KUKA KRL program: Robotarmmovement.src

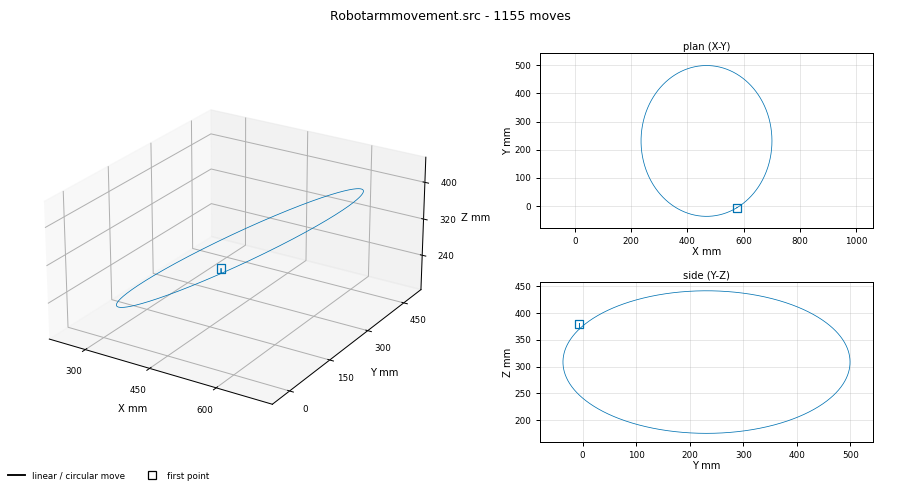
[picture p0: tool path of Robotarmmovement.src, 1155 of 1157 moves have a stored position in this frame; points joined in program order, loops and branches not executed]
&ACCESS RVP
&PARAM EDITMASK = *
&PARAM TEMPLATE = C:\KRC\Roboter\Template\vorgabe
DEF Robotarmmovement( )


;FOLD INI
;FOLD BASISTECH INI
GLOBAL INTERRUPT DECL 3 WHEN $STOPMESS==TRUE DO IR_STOPM ( )
INTERRUPT ON 3
BAS (#INITMOV,0 )
;ENDFOLD (BASISTECH INI)
;ENDFOLD (INI)

;FOLD STARTPOSITION - BASE IS 0, TOOL IS 6, SPEED IS 15%, POSITION IS A1 5,A2 -90,A3 100,A4 5,A5 -10,A6 -5,E1 0,E2 0,E3 0,E4 0
$BWDSTART = FALSE
PDAT_ACT = {VEL 15,ACC 100,APO_DIST 50}
FDAT_ACT = {TOOL_NO 6,BASE_NO 0,IPO_FRAME #BASE}
BAS (#PTP_PARAMS,15)
PTP  {A1 5,A2 -90,A3 100,A4 5,A5 -10,A6 -5,E1 0,E2 0,E3 0,E4 0}
;ENDFOLD

;FOLD LIN SPEED IS 0.25 m/sec, INTERPOLATION SETTINGS IN FOLD
$VEL.CP=0.25
$ADVANCE=3
;ENDFOLD

;FOLD COMMANDS IN FOLD. SELECT EDIT/FOLDS/OPEN ALL FOLDS TO DISPLAY
PTP {X 576.159, Y -6.053, Z 380.301, A 0, B 90, C -61.802, E1 0, E2 0, E3 0, E4 0, S 'B 110'} C_PTP
LIN {X 576.159, Y -6.053, Z 380.301, A 0, B 90, C -61.802, E1 0, E2 0, E3 0, E4 0}
LIN {X 576.159, Y -6.053, Z 370.301, A 0, B 90, C -61.802, E1 0, E2 0, E3 0, E4 0} C_DIS
LIN {X 577.282, Y -5.37, Z 370.943, A 0, B 90, C -61.726, E1 0, E2 0, E3 0, E4 0} C_DIS
LIN {X 578.402, Y -4.68, Z 371.584, A 0, B 90, C -61.652, E1 0, E2 0, E3 0, E4 0} C_DIS
LIN {X 579.519, Y -3.984, Z 372.223, A 0, B 90, C -61.578, E1 0, E2 0, E3 0, E4 0} C_DIS
LIN {X 580.632, Y -3.28, Z 372.86, A 0, B 90, C -61.506, E1 0, E2 0, E3 0, E4 0} C_DIS
LIN {X 581.742, Y -2.569, Z 373.495, A 0, B 90, C -61.434, E1 0, E2 0, E3 0, E4 0} C_DIS
LIN {X 582.848, Y -1.851, Z 374.128, A 0, B 90, C -61.364, E1 0, E2 0, E3 0, E4 0} C_DIS
LIN {X 583.952, Y -1.126, Z 374.759, A 0, B 90, C -61.294, E1 0, E2 0, E3 0, E4 0} C_DIS
LIN {X 585.051, Y -0.395, Z 375.389, A 0, B 90, C -61.226, E1 0, E2 0, E3 0, E4 0} C_DIS
LIN {X 586.148, Y 0.344, Z 376.016, A 0, B 90, C -61.159, E1 0, E2 0, E3 0, E4 0} C_DIS
LIN {X 587.24, Y 1.089, Z 376.641, A 0, B 90, C -61.093, E1 0, E2 0, E3 0, E4 0} C_DIS
LIN {X 588.329, Y 1.842, Z 377.264, A 0, B 90, C -61.027, E1 0, E2 0, E3 0, E4 0} C_DIS
LIN {X 589.415, Y 2.601, Z 377.885, A 0, B 90, C -60.963, E1 0, E2 0, E3 0, E4 0} C_DIS
LIN {X 590.497, Y 3.367, Z 378.504, A 0, B 90, C -60.9, E1 0, E2 0, E3 0, E4 0} C_DIS
LIN {X 591.575, Y 4.14, Z 379.121, A 0, B 90, C -60.838, E1 0, E2 0, E3 0, E4 0} C_DIS
LIN {X 592.65, Y 4.919, Z 379.736, A 0, B 90, C -60.776, E1 0, E2 0, E3 0, E4 0} C_DIS
LIN {X 593.721, Y 5.705, Z 380.349, A 0, B 90, C -60.716, E1 0, E2 0, E3 0, E4 0} C_DIS
LIN {X 594.788, Y 6.498, Z 380.96, A 0, B 90, C -60.657, E1 0, E2 0, E3 0, E4 0} C_DIS
LIN {X 595.851, Y 7.298, Z 381.568, A 0, B 90, C -60.598, E1 0, E2 0, E3 0, E4 0} C_DIS
LIN {X 596.911, Y 8.105, Z 382.174, A 0, B 90, C -60.541, E1 0, E2 0, E3 0, E4 0} C_DIS
LIN {X 597.967, Y 8.918, Z 382.778, A 0, B 90, C -60.485, E1 0, E2 0, E3 0, E4 0} C_DIS
LIN {X 599.019, Y 9.737, Z 383.38, A 0, B 90, C -60.43, E1 0, E2 0, E3 0, E4 0} C_DIS
LIN {X 600.067, Y 10.564, Z 383.98, A 0, B 90, C -60.375, E1 0, E2 0, E3 0, E4 0} C_DIS
LIN {X 601.111, Y 11.396, Z 384.577, A 0, B 90, C -60.322, E1 0, E2 0, E3 0, E4 0} C_DIS
LIN {X 602.151, Y 12.236, Z 385.172, A 0, B 90, C -60.269, E1 0, E2 0, E3 0, E4 0} C_DIS
LIN {X 603.187, Y 13.082, Z 385.765, A 0, B 90, C -60.218, E1 0, E2 0, E3 0, E4 0} C_DIS
LIN {X 604.219, Y 13.934, Z 386.356, A 0, B 90, C -60.167, E1 0, E2 0, E3 0, E4 0} C_DIS
LIN {X 605.247, Y 14.793, Z 386.944, A 0, B 90, C -60.118, E1 0, E2 0, E3 0, E4 0} C_DIS
LIN {X 606.271, Y 15.658, Z 387.53, A 0, B 90, C -60.069, E1 0, E2 0, E3 0, E4 0} C_DIS
LIN {X 607.291, Y 16.53, Z 388.113, A 0, B 90, C -60.022, E1 0, E2 0, E3 0, E4 0} C_DIS
LIN {X 608.307, Y 17.408, Z 388.695, A 0, B 90, C -59.975, E1 0, E2 0, E3 0, E4 0} C_DIS
LIN {X 609.318, Y 18.293, Z 389.273, A 0, B 90, C -59.929, E1 0, E2 0, E3 0, E4 0} C_DIS
LIN {X 610.325, Y 19.184, Z 389.85, A 0, B 90, C -59.884, E1 0, E2 0, E3 0, E4 0} C_DIS
LIN {X 611.328, Y 20.081, Z 390.424, A 0, B 90, C -59.84, E1 0, E2 0, E3 0, E4 0} C_DIS
LIN {X 612.327, Y 20.985, Z 390.995, A 0, B 90, C -59.798, E1 0, E2 0, E3 0, E4 0} C_DIS
LIN {X 613.322, Y 21.895, Z 391.564, A 0, B 90, C -59.755, E1 0, E2 0, E3 0, E4 0} C_DIS
LIN {X 614.312, Y 22.811, Z 392.131, A 0, B 90, C -59.714, E1 0, E2 0, E3 0, E4 0} C_DIS
LIN {X 615.298, Y 23.733, Z 392.695, A 0, B 90, C -59.674, E1 0, E2 0, E3 0, E4 0} C_DIS
LIN {X 616.279, Y 24.661, Z 393.256, A 0, B 90, C -59.635, E1 0, E2 0, E3 0, E4 0} C_DIS
LIN {X 617.256, Y 25.596, Z 393.815, A 0, B 90, C -59.596, E1 0, E2 0, E3 0, E4 0} C_DIS
LIN {X 618.229, Y 26.537, Z 394.372, A 0, B 90, C -59.559, E1 0, E2 0, E3 0, E4 0} C_DIS
LIN {X 619.197, Y 27.483, Z 394.926, A 0, B 90, C -59.522, E1 0, E2 0, E3 0, E4 0} C_DIS
LIN {X 620.161, Y 28.436, Z 395.477, A 0, B 90, C -59.486, E1 0, E2 0, E3 0, E4 0} C_DIS
LIN {X 621.12, Y 29.395, Z 396.026, A 0, B 90, C -59.452, E1 0, E2 0, E3 0, E4 0} C_DIS
LIN {X 622.074, Y 30.36, Z 396.572, A 0, B 90, C -59.418, E1 0, E2 0, E3 0, E4 0} C_DIS
LIN {X 623.024, Y 31.331, Z 397.116, A 0, B 90, C -59.385, E1 0, E2 0, E3 0, E4 0} C_DIS
LIN {X 623.97, Y 32.308, Z 397.657, A 0, B 90, C -59.352, E1 0, E2 0, E3 0, E4 0} C_DIS
LIN {X 624.91, Y 33.291, Z 398.195, A 0, B 90, C -59.321, E1 0, E2 0, E3 0, E4 0} C_DIS
LIN {X 625.846, Y 34.28, Z 398.73, A 0, B 90, C -59.29, E1 0, E2 0, E3 0, E4 0} C_DIS
LIN {X 626.778, Y 35.274, Z 399.263, A 0, B 90, C -59.261, E1 0, E2 0, E3 0, E4 0} C_DIS
LIN {X 627.704, Y 36.275, Z 399.793, A 0, B 90, C -59.232, E1 0, E2 0, E3 0, E4 0} C_DIS
LIN {X 628.626, Y 37.281, Z 400.321, A 0, B 90, C -59.204, E1 0, E2 0, E3 0, E4 0} C_DIS
LIN {X 629.543, Y 38.293, Z 400.846, A 0, B 90, C -59.177, E1 0, E2 0, E3 0, E4 0} C_DIS
LIN {X 630.455, Y 39.311, Z 401.368, A 0, B 90, C -59.151, E1 0, E2 0, E3 0, E4 0} C_DIS
LIN {X 631.363, Y 40.335, Z 401.887, A 0, B 90, C -59.125, E1 0, E2 0, E3 0, E4 0} C_DIS
LIN {X 632.265, Y 41.364, Z 402.403, A 0, B 90, C -59.101, E1 0, E2 0, E3 0, E4 0} C_DIS
LIN {X 633.163, Y 42.399, Z 402.917, A 0, B 90, C -59.077, E1 0, E2 0, E3 0, E4 0} C_DIS
LIN {X 634.056, Y 43.439, Z 403.428, A 0, B 90, C -59.054, E1 0, E2 0, E3 0, E4 0} C_DIS
LIN {X 634.943, Y 44.485, Z 403.936, A 0, B 90, C -59.032, E1 0, E2 0, E3 0, E4 0} C_DIS
LIN {X 635.826, Y 45.537, Z 404.441, A 0, B 90, C -59.01, E1 0, E2 0, E3 0, E4 0} C_DIS
LIN {X 636.704, Y 46.594, Z 404.943, A 0, B 90, C -58.99, E1 0, E2 0, E3 0, E4 0} C_DIS
LIN {X 637.577, Y 47.657, Z 405.442, A 0, B 90, C -58.97, E1 0, E2 0, E3 0, E4 0} C_DIS
LIN {X 638.445, Y 48.725, Z 405.939, A 0, B 90, C -58.951, E1 0, E2 0, E3 0, E4 0} C_DIS
LIN {X 639.307, Y 49.799, Z 406.432, A 0, B 90, C -58.933, E1 0, E2 0, E3 0, E4 0} C_DIS
LIN {X 640.165, Y 50.878, Z 406.923, A 0, B 90, C -58.916, E1 0, E2 0, E3 0, E4 0} C_DIS
LIN {X 641.017, Y 51.962, Z 407.411, A 0, B 90, C -58.899, E1 0, E2 0, E3 0, E4 0} C_DIS
LIN {X 641.865, Y 53.052, Z 407.896, A 0, B 90, C -58.883, E1 0, E2 0, E3 0, E4 0} C_DIS
LIN {X 642.707, Y 54.147, Z 408.378, A 0, B 90, C -58.868, E1 0, E2 0, E3 0, E4 0} C_DIS
LIN {X 643.544, Y 55.248, Z 408.856, A 0, B 90, C -58.854, E1 0, E2 0, E3 0, E4 0} C_DIS
LIN {X 644.375, Y 56.353, Z 409.332, A 0, B 90, C -58.84, E1 0, E2 0, E3 0, E4 0} C_DIS
LIN {X 645.202, Y 57.464, Z 409.805, A 0, B 90, C -58.828, E1 0, E2 0, E3 0, E4 0} C_DIS
LIN {X 646.023, Y 58.58, Z 410.275, A 0, B 90, C -58.816, E1 0, E2 0, E3 0, E4 0} C_DIS
LIN {X 646.839, Y 59.701, Z 410.742, A 0, B 90, C -58.804, E1 0, E2 0, E3 0, E4 0} C_DIS
LIN {X 647.65, Y 60.828, Z 411.206, A 0, B 90, C -58.794, E1 0, E2 0, E3 0, E4 0} C_DIS
LIN {X 648.455, Y 61.959, Z 411.666, A 0, B 90, C -58.784, E1 0, E2 0, E3 0, E4 0} C_DIS
LIN {X 649.255, Y 63.095, Z 412.124, A 0, B 90, C -58.775, E1 0, E2 0, E3 0, E4 0} C_DIS
LIN {X 650.049, Y 64.237, Z 412.579, A 0, B 90, C -58.767, E1 0, E2 0, E3 0, E4 0} C_DIS
LIN {X 650.838, Y 65.383, Z 413.03, A 0, B 90, C -58.759, E1 0, E2 0, E3 0, E4 0} C_DIS
LIN {X 651.622, Y 66.535, Z 413.478, A 0, B 90, C -58.752, E1 0, E2 0, E3 0, E4 0} C_DIS
LIN {X 652.4, Y 67.691, Z 413.924, A 0, B 90, C -58.746, E1 0, E2 0, E3 0, E4 0} C_DIS
LIN {X 653.172, Y 68.852, Z 414.366, A 0, B 90, C -58.74, E1 0, E2 0, E3 0, E4 0} C_DIS
LIN {X 653.94, Y 70.018, Z 414.805, A 0, B 90, C -58.736, E1 0, E2 0, E3 0, E4 0} C_DIS
LIN {X 654.701, Y 71.189, Z 415.24, A 0, B 90, C -58.732, E1 0, E2 0, E3 0, E4 0} C_DIS
LIN {X 655.457, Y 72.364, Z 415.673, A 0, B 90, C -58.728, E1 0, E2 0, E3 0, E4 0} C_DIS
LIN {X 656.208, Y 73.545, Z 416.102, A 0, B 90, C -58.726, E1 0, E2 0, E3 0, E4 0} C_DIS
LIN {X 656.952, Y 74.73, Z 416.529, A 0, B 90, C -58.724, E1 0, E2 0, E3 0, E4 0} C_DIS
LIN {X 657.692, Y 75.919, Z 416.951, A 0, B 90, C -58.722, E1 0, E2 0, E3 0, E4 0} C_DIS
LIN {X 658.425, Y 77.114, Z 417.371, A 0, B 90, C -58.722, E1 0, E2 0, E3 0, E4 0} C_DIS
LIN {X 659.153, Y 78.313, Z 417.788, A 0, B 90, C -58.722, E1 0, E2 0, E3 0, E4 0} C_DIS
LIN {X 659.875, Y 79.516, Z 418.201, A 0, B 90, C -58.722, E1 0, E2 0, E3 0, E4 0} C_DIS
LIN {X 660.592, Y 80.724, Z 418.611, A 0, B 90, C -58.724, E1 0, E2 0, E3 0, E4 0} C_DIS
LIN {X 661.302, Y 81.936, Z 419.017, A 0, B 90, C -58.726, E1 0, E2 0, E3 0, E4 0} C_DIS
LIN {X 662.007, Y 83.153, Z 419.421, A 0, B 90, C -58.728, E1 0, E2 0, E3 0, E4 0} C_DIS
LIN {X 662.707, Y 84.375, Z 419.821, A 0, B 90, C -58.732, E1 0, E2 0, E3 0, E4 0} C_DIS
LIN {X 663.4, Y 85.6, Z 420.218, A 0, B 90, C -58.736, E1 0, E2 0, E3 0, E4 0} C_DIS
LIN {X 664.088, Y 86.83, Z 420.611, A 0, B 90, C -58.74, E1 0, E2 0, E3 0, E4 0} C_DIS
LIN {X 664.769, Y 88.065, Z 421.001, A 0, B 90, C -58.746, E1 0, E2 0, E3 0, E4 0} C_DIS
LIN {X 665.445, Y 89.303, Z 421.388, A 0, B 90, C -58.751, E1 0, E2 0, E3 0, E4 0} C_DIS
LIN {X 666.115, Y 90.546, Z 421.771, A 0, B 90, C -58.758, E1 0, E2 0, E3 0, E4 0} C_DIS
LIN {X 666.779, Y 91.793, Z 422.151, A 0, B 90, C -58.765, E1 0, E2 0, E3 0, E4 0} C_DIS
LIN {X 667.438, Y 93.045, Z 422.528, A 0, B 90, C -58.773, E1 0, E2 0, E3 0, E4 0} C_DIS
LIN {X 668.09, Y 94.3, Z 422.901, A 0, B 90, C -58.781, E1 0, E2 0, E3 0, E4 0} C_DIS
LIN {X 668.736, Y 95.559, Z 423.271, A 0, B 90, C -58.79, E1 0, E2 0, E3 0, E4 0} C_DIS
LIN {X 669.376, Y 96.823, Z 423.637, A 0, B 90, C -58.8, E1 0, E2 0, E3 0, E4 0} C_DIS
LIN {X 670.011, Y 98.09, Z 424, A 0, B 90, C -58.81, E1 0, E2 0, E3 0, E4 0} C_DIS
LIN {X 670.639, Y 99.362, Z 424.36, A 0, B 90, C -58.821, E1 0, E2 0, E3 0, E4 0} C_DIS
LIN {X 671.261, Y 100.637, Z 424.716, A 0, B 90, C -58.832, E1 0, E2 0, E3 0, E4 0} C_DIS
LIN {X 671.878, Y 101.916, Z 425.068, A 0, B 90, C -58.844, E1 0, E2 0, E3 0, E4 0} C_DIS
LIN {X 672.488, Y 103.199, Z 425.418, A 0, B 90, C -58.856, E1 0, E2 0, E3 0, E4 0} C_DIS
LIN {X 673.092, Y 104.486, Z 425.763, A 0, B 90, C -58.87, E1 0, E2 0, E3 0, E4 0} C_DIS
LIN {X 673.69, Y 105.777, Z 426.105, A 0, B 90, C -58.883, E1 0, E2 0, E3 0, E4 0} C_DIS
LIN {X 674.282, Y 107.072, Z 426.444, A 0, B 90, C -58.898, E1 0, E2 0, E3 0, E4 0} C_DIS
LIN {X 674.867, Y 108.37, Z 426.779, A 0, B 90, C -58.912, E1 0, E2 0, E3 0, E4 0} C_DIS
LIN {X 675.447, Y 109.672, Z 427.111, A 0, B 90, C -58.928, E1 0, E2 0, E3 0, E4 0} C_DIS
LIN {X 676.02, Y 110.977, Z 427.439, A 0, B 90, C -58.944, E1 0, E2 0, E3 0, E4 0} C_DIS
LIN {X 676.588, Y 112.286, Z 427.763, A 0, B 90, C -58.96, E1 0, E2 0, E3 0, E4 0} C_DIS
LIN {X 677.148, Y 113.599, Z 428.084, A 0, B 90, C -58.977, E1 0, E2 0, E3 0, E4 0} C_DIS
LIN {X 677.703, Y 114.915, Z 428.402, A 0, B 90, C -58.995, E1 0, E2 0, E3 0, E4 0} C_DIS
LIN {X 678.252, Y 116.234, Z 428.715, A 0, B 90, C -59.013, E1 0, E2 0, E3 0, E4 0} C_DIS
LIN {X 678.794, Y 117.557, Z 429.026, A 0, B 90, C -59.032, E1 0, E2 0, E3 0, E4 0} C_DIS
LIN {X 679.33, Y 118.884, Z 429.332, A 0, B 90, C -59.051, E1 0, E2 0, E3 0, E4 0} C_DIS
LIN {X 679.859, Y 120.214, Z 429.635, A 0, B 90, C -59.071, E1 0, E2 0, E3 0, E4 0} C_DIS
LIN {X 680.383, Y 121.547, Z 429.935, A 0, B 90, C -59.091, E1 0, E2 0, E3 0, E4 0} C_DIS
LIN {X 680.9, Y 122.883, Z 430.231, A 0, B 90, C -59.112, E1 0, E2 0, E3 0, E4 0} C_DIS
LIN {X 681.411, Y 124.222, Z 430.523, A 0, B 90, C -59.133, E1 0, E2 0, E3 0, E4 0} C_DIS
LIN {X 681.915, Y 125.565, Z 430.811, A 0, B 90, C -59.155, E1 0, E2 0, E3 0, E4 0} C_DIS
LIN {X 682.413, Y 126.911, Z 431.096, A 0, B 90, C -59.177, E1 0, E2 0, E3 0, E4 0} C_DIS
LIN {X 682.904, Y 128.26, Z 431.378, A 0, B 90, C -59.2, E1 0, E2 0, E3 0, E4 0} C_DIS
LIN {X 683.39, Y 129.612, Z 431.655, A 0, B 90, C -59.224, E1 0, E2 0, E3 0, E4 0} C_DIS
LIN {X 683.868, Y 130.967, Z 431.929, A 0, B 90, C -59.247, E1 0, E2 0, E3 0, E4 0} C_DIS
LIN {X 684.341, Y 132.325, Z 432.199, A 0, B 90, C -59.272, E1 0, E2 0, E3 0, E4 0} C_DIS
LIN {X 684.807, Y 133.687, Z 432.466, A 0, B 90, C -59.297, E1 0, E2 0, E3 0, E4 0} C_DIS
LIN {X 685.266, Y 135.051, Z 432.729, A 0, B 90, C -59.322, E1 0, E2 0, E3 0, E4 0} C_DIS
LIN {X 685.719, Y 136.417, Z 432.988, A 0, B 90, C -59.348, E1 0, E2 0, E3 0, E4 0} C_DIS
LIN {X 686.166, Y 137.787, Z 433.244, A 0, B 90, C -59.374, E1 0, E2 0, E3 0, E4 0} C_DIS
LIN {X 686.606, Y 139.159, Z 433.495, A 0, B 90, C -59.401, E1 0, E2 0, E3 0, E4 0} C_DIS
LIN {X 687.039, Y 140.535, Z 433.743, A 0, B 90, C -59.428, E1 0, E2 0, E3 0, E4 0} C_DIS
LIN {X 687.466, Y 141.913, Z 433.988, A 0, B 90, C -59.456, E1 0, E2 0, E3 0, E4 0} C_DIS
LIN {X 687.886, Y 143.293, Z 434.228, A 0, B 90, C -59.484, E1 0, E2 0, E3 0, E4 0} C_DIS
LIN {X 688.3, Y 144.676, Z 434.465, A 0, B 90, C -59.513, E1 0, E2 0, E3 0, E4 0} C_DIS
LIN {X 688.708, Y 146.062, Z 434.698, A 0, B 90, C -59.542, E1 0, E2 0, E3 0, E4 0} C_DIS
LIN {X 689.108, Y 147.45, Z 434.927, A 0, B 90, C -59.571, E1 0, E2 0, E3 0, E4 0} C_DIS
LIN {X 689.503, Y 148.841, Z 435.153, A 0, B 90, C -59.601, E1 0, E2 0, E3 0, E4 0} C_DIS
LIN {X 689.89, Y 150.235, Z 435.375, A 0, B 90, C -59.632, E1 0, E2 0, E3 0, E4 0} C_DIS
LIN {X 690.271, Y 151.63, Z 435.593, A 0, B 90, C -59.663, E1 0, E2 0, E3 0, E4 0} C_DIS
LIN {X 690.645, Y 153.028, Z 435.807, A 0, B 90, C -59.694, E1 0, E2 0, E3 0, E4 0} C_DIS
LIN {X 691.013, Y 154.429, Z 436.017, A 0, B 90, C -59.726, E1 0, E2 0, E3 0, E4 0} C_DIS
LIN {X 691.374, Y 155.831, Z 436.224, A 0, B 90, C -59.758, E1 0, E2 0, E3 0, E4 0} C_DIS
LIN {X 691.729, Y 157.236, Z 436.427, A 0, B 90, C -59.791, E1 0, E2 0, E3 0, E4 0} C_DIS
LIN {X 692.076, Y 158.643, Z 436.626, A 0, B 90, C -59.824, E1 0, E2 0, E3 0, E4 0} C_DIS
LIN {X 692.417, Y 160.053, Z 436.821, A 0, B 90, C -59.858, E1 0, E2 0, E3 0, E4 0} C_DIS
LIN {X 692.752, Y 161.464, Z 437.012, A 0, B 90, C -59.892, E1 0, E2 0, E3 0, E4 0} C_DIS
LIN {X 693.08, Y 162.878, Z 437.2, A 0, B 90, C -59.926, E1 0, E2 0, E3 0, E4 0} C_DIS
LIN {X 693.401, Y 164.293, Z 437.383, A 0, B 90, C -59.961, E1 0, E2 0, E3 0, E4 0} C_DIS
LIN {X 693.715, Y 165.711, Z 437.563, A 0, B 90, C -59.996, E1 0, E2 0, E3 0, E4 0} C_DIS
LIN {X 694.022, Y 167.13, Z 437.739, A 0, B 90, C -60.032, E1 0, E2 0, E3 0, E4 0} C_DIS
LIN {X 694.323, Y 168.552, Z 437.911, A 0, B 90, C -60.068, E1 0, E2 0, E3 0, E4 0} C_DIS
LIN {X 694.617, Y 169.975, Z 438.079, A 0, B 90, C -60.104, E1 0, E2 0, E3 0, E4 0} C_DIS
LIN {X 694.905, Y 171.4, Z 438.244, A 0, B 90, C -60.141, E1 0, E2 0, E3 0, E4 0} C_DIS
LIN {X 695.185, Y 172.827, Z 438.404, A 0, B 90, C -60.178, E1 0, E2 0, E3 0, E4 0} C_DIS
LIN {X 695.459, Y 174.256, Z 438.561, A 0, B 90, C -60.216, E1 0, E2 0, E3 0, E4 0} C_DIS
LIN {X 695.726, Y 175.686, Z 438.714, A 0, B 90, C -60.254, E1 0, E2 0, E3 0, E4 0} C_DIS
LIN {X 695.987, Y 177.118, Z 438.863, A 0, B 90, C -60.292, E1 0, E2 0, E3 0, E4 0} C_DIS
LIN {X 696.24, Y 178.552, Z 439.008, A 0, B 90, C -60.331, E1 0, E2 0, E3 0, E4 0} C_DIS
LIN {X 696.487, Y 179.987, Z 439.149, A 0, B 90, C -60.37, E1 0, E2 0, E3 0, E4 0} C_DIS
LIN {X 696.727, Y 181.424, Z 439.286, A 0, B 90, C -60.409, E1 0, E2 0, E3 0, E4 0} C_DIS
LIN {X 696.96, Y 182.862, Z 439.42, A 0, B 90, C -60.449, E1 0, E2 0, E3 0, E4 0} C_DIS
LIN {X 697.186, Y 184.302, Z 439.549, A 0, B 90, C -60.49, E1 0, E2 0, E3 0, E4 0} C_DIS
LIN {X 697.405, Y 185.743, Z 439.675, A 0, B 90, C -60.53, E1 0, E2 0, E3 0, E4 0} C_DIS
LIN {X 697.618, Y 187.185, Z 439.796, A 0, B 90, C -60.571, E1 0, E2 0, E3 0, E4 0} C_DIS
LIN {X 697.824, Y 188.629, Z 439.914, A 0, B 90, C -60.613, E1 0, E2 0, E3 0, E4 0} C_DIS
LIN {X 698.023, Y 190.074, Z 440.028, A 0, B 90, C -60.654, E1 0, E2 0, E3 0, E4 0} C_DIS
LIN {X 698.215, Y 191.52, Z 440.138, A 0, B 90, C -60.696, E1 0, E2 0, E3 0, E4 0} C_DIS
LIN {X 698.4, Y 192.968, Z 440.244, A 0, B 90, C -60.739, E1 0, E2 0, E3 0, E4 0} C_DIS
LIN {X 698.578, Y 194.416, Z 440.346, A 0, B 90, C -60.782, E1 0, E2 0, E3 0, E4 0} C_DIS
LIN {X 698.75, Y 195.866, Z 440.444, A 0, B 90, C -60.825, E1 0, E2 0, E3 0, E4 0} C_DIS
LIN {X 698.914, Y 197.317, Z 440.538, A 0, B 90, C -60.868, E1 0, E2 0, E3 0, E4 0} C_DIS
LIN {X 699.072, Y 198.768, Z 440.628, A 0, B 90, C -60.912, E1 0, E2 0, E3 0, E4 0} C_DIS
LIN {X 699.223, Y 200.221, Z 440.715, A 0, B 90, C -60.956, E1 0, E2 0, E3 0, E4 0} C_DIS
LIN {X 699.367, Y 201.675, Z 440.797, A 0, B 90, C -61.001, E1 0, E2 0, E3 0, E4 0} C_DIS
LIN {X 699.504, Y 203.129, Z 440.876, A 0, B 90, C -61.046, E1 0, E2 0, E3 0, E4 0} C_DIS
LIN {X 699.634, Y 204.585, Z 440.95, A 0, B 90, C -61.091, E1 0, E2 0, E3 0, E4 0} C_DIS
LIN {X 699.758, Y 206.041, Z 441.021, A 0, B 90, C -61.136, E1 0, E2 0, E3 0, E4 0} C_DIS
LIN {X 699.874, Y 207.498, Z 441.087, A 0, B 90, C -61.182, E1 0, E2 0, E3 0, E4 0} C_DIS
LIN {X 699.983, Y 208.955, Z 441.15, A 0, B 90, C -61.228, E1 0, E2 0, E3 0, E4 0} C_DIS
LIN {X 700.086, Y 210.414, Z 441.209, A 0, B 90, C -61.275, E1 0, E2 0, E3 0, E4 0} C_DIS
LIN {X 700.182, Y 211.873, Z 441.263, A 0, B 90, C -61.322, E1 0, E2 0, E3 0, E4 0} C_DIS
LIN {X 700.271, Y 213.332, Z 441.314, A 0, B 90, C -61.369, E1 0, E2 0, E3 0, E4 0} C_DIS
LIN {X 700.352, Y 214.792, Z 441.361, A 0, B 90, C -61.416, E1 0, E2 0, E3 0, E4 0} C_DIS
LIN {X 700.427, Y 216.253, Z 441.404, A 0, B 90, C -61.464, E1 0, E2 0, E3 0, E4 0} C_DIS
LIN {X 700.495, Y 217.714, Z 441.443, A 0, B 90, C -61.512, E1 0, E2 0, E3 0, E4 0} C_DIS
LIN {X 700.556, Y 219.175, Z 441.478, A 0, B 90, C -61.56, E1 0, E2 0, E3 0, E4 0} C_DIS
LIN {X 700.61, Y 220.637, Z 441.509, A 0, B 90, C -61.609, E1 0, E2 0, E3 0, E4 0} C_DIS
LIN {X 700.658, Y 222.099, Z 441.536, A 0, B 90, C -61.658, E1 0, E2 0, E3 0, E4 0} C_DIS
LIN {X 700.698, Y 223.561, Z 441.559, A 0, B 90, C -61.707, E1 0, E2 0, E3 0, E4 0} C_DIS
LIN {X 700.731, Y 225.024, Z 441.578, A 0, B 90, C -61.757, E1 0, E2 0, E3 0, E4 0} C_DIS
LIN {X 700.758, Y 226.487, Z 441.593, A 0, B 90, C -61.807, E1 0, E2 0, E3 0, E4 0} C_DIS
LIN {X 700.777, Y 227.95, Z 441.604, A 0, B 90, C -61.857, E1 0, E2 0, E3 0, E4 0} C_DIS
LIN {X 700.79, Y 229.413, Z 441.611, A 0, B 90, C -61.907, E1 0, E2 0, E3 0, E4 0} C_DIS
LIN {X 700.796, Y 230.876, Z 441.614, A 0, B 90, C -61.958, E1 0, E2 0, E3 0, E4 0} C_DIS
LIN {X 700.794, Y 232.339, Z 441.614, A 0, B 90, C -62.009, E1 0, E2 0, E3 0, E4 0} C_DIS
LIN {X 700.786, Y 233.802, Z 441.609, A 0, B 90, C -62.06, E1 0, E2 0, E3 0, E4 0} C_DIS
LIN {X 700.771, Y 235.265, Z 441.6, A 0, B 90, C -62.112, E1 0, E2 0, E3 0, E4 0} C_DIS
LIN {X 700.749, Y 236.728, Z 441.588, A 0, B 90, C -62.164, E1 0, E2 0, E3 0, E4 0} C_DIS
LIN {X 700.72, Y 238.19, Z 441.571, A 0, B 90, C -62.216, E1 0, E2 0, E3 0, E4 0} C_DIS
LIN {X 700.684, Y 239.653, Z 441.551, A 0, B 90, C -62.268, E1 0, E2 0, E3 0, E4 0} C_DIS
LIN {X 700.641, Y 241.115, Z 441.526, A 0, B 90, C -62.321, E1 0, E2 0, E3 0, E4 0} C_DIS
LIN {X 700.591, Y 242.577, Z 441.498, A 0, B 90, C -62.374, E1 0, E2 0, E3 0, E4 0} C_DIS
LIN {X 700.534, Y 244.039, Z 441.465, A 0, B 90, C -62.427, E1 0, E2 0, E3 0, E4 0} C_DIS
LIN {X 700.471, Y 245.5, Z 441.429, A 0, B 90, C -62.481, E1 0, E2 0, E3 0, E4 0} C_DIS
LIN {X 700.4, Y 246.961, Z 441.388, A 0, B 90, C -62.534, E1 0, E2 0, E3 0, E4 0} C_DIS
LIN {X 700.323, Y 248.421, Z 441.344, A 0, B 90, C -62.588, E1 0, E2 0, E3 0, E4 0} C_DIS
LIN {X 700.238, Y 249.881, Z 441.296, A 0, B 90, C -62.643, E1 0, E2 0, E3 0, E4 0} C_DIS
LIN {X 700.147, Y 251.34, Z 441.243, A 0, B 90, C -62.697, E1 0, E2 0, E3 0, E4 0} C_DIS
LIN {X 700.049, Y 252.799, Z 441.187, A 0, B 90, C -62.752, E1 0, E2 0, E3 0, E4 0} C_DIS
LIN {X 699.943, Y 254.257, Z 441.127, A 0, B 90, C -62.807, E1 0, E2 0, E3 0, E4 0} C_DIS
LIN {X 699.832, Y 255.714, Z 441.063, A 0, B 90, C -62.862, E1 0, E2 0, E3 0, E4 0} C_DIS
LIN {X 699.713, Y 257.171, Z 440.995, A 0, B 90, C -62.917, E1 0, E2 0, E3 0, E4 0} C_DIS
LIN {X 699.587, Y 258.627, Z 440.923, A 0, B 90, C -62.973, E1 0, E2 0, E3 0, E4 0} C_DIS
LIN {X 699.454, Y 260.082, Z 440.847, A 0, B 90, C -63.029, E1 0, E2 0, E3 0, E4 0} C_DIS
LIN {X 699.314, Y 261.536, Z 440.767, A 0, B 90, C -63.085, E1 0, E2 0, E3 0, E4 0} C_DIS
LIN {X 699.168, Y 262.989, Z 440.683, A 0, B 90, C -63.142, E1 0, E2 0, E3 0, E4 0} C_DIS
LIN {X 699.014, Y 264.442, Z 440.595, A 0, B 90, C -63.198, E1 0, E2 0, E3 0, E4 0} C_DIS
LIN {X 698.854, Y 265.893, Z 440.504, A 0, B 90, C -63.255, E1 0, E2 0, E3 0, E4 0} C_DIS
LIN {X 698.687, Y 267.343, Z 440.408, A 0, B 90, C -63.313, E1 0, E2 0, E3 0, E4 0} C_DIS
LIN {X 698.513, Y 268.793, Z 440.308, A 0, B 90, C -63.37, E1 0, E2 0, E3 0, E4 0} C_DIS
LIN {X 698.332, Y 270.241, Z 440.205, A 0, B 90, C -63.428, E1 0, E2 0, E3 0, E4 0} C_DIS
LIN {X 698.144, Y 271.688, Z 440.097, A 0, B 90, C -63.485, E1 0, E2 0, E3 0, E4 0} C_DIS
LIN {X 697.95, Y 273.134, Z 439.986, A 0, B 90, C -63.543, E1 0, E2 0, E3 0, E4 0} C_DIS
LIN {X 697.748, Y 274.578, Z 439.871, A 0, B 90, C -63.602, E1 0, E2 0, E3 0, E4 0} C_DIS
LIN {X 697.54, Y 276.021, Z 439.752, A 0, B 90, C -63.66, E1 0, E2 0, E3 0, E4 0} C_DIS
LIN {X 697.325, Y 277.463, Z 439.628, A 0, B 90, C -63.719, E1 0, E2 0, E3 0, E4 0} C_DIS
LIN {X 697.103, Y 278.904, Z 439.501, A 0, B 90, C -63.778, E1 0, E2 0, E3 0, E4 0} C_DIS
LIN {X 696.874, Y 280.343, Z 439.371, A 0, B 90, C -63.837, E1 0, E2 0, E3 0, E4 0} C_DIS
LIN {X 696.638, Y 281.781, Z 439.236, A 0, B 90, C -63.896, E1 0, E2 0, E3 0, E4 0} C_DIS
LIN {X 696.396, Y 283.217, Z 439.097, A 0, B 90, C -63.956, E1 0, E2 0, E3 0, E4 0} C_DIS
LIN {X 696.147, Y 284.652, Z 438.954, A 0, B 90, C -64.016, E1 0, E2 0, E3 0, E4 0} C_DIS
LIN {X 695.891, Y 286.085, Z 438.808, A 0, B 90, C -64.076, E1 0, E2 0, E3 0, E4 0} C_DIS
LIN {X 695.628, Y 287.516, Z 438.658, A 0, B 90, C -64.136, E1 0, E2 0, E3 0, E4 0} C_DIS
LIN {X 695.358, Y 288.946, Z 438.503, A 0, B 90, C -64.196, E1 0, E2 0, E3 0, E4 0} C_DIS
LIN {X 695.082, Y 290.374, Z 438.345, A 0, B 90, C -64.257, E1 0, E2 0, E3 0, E4 0} C_DIS
LIN {X 694.799, Y 291.8, Z 438.183, A 0, B 90, C -64.318, E1 0, E2 0, E3 0, E4 0} C_DIS
LIN {X 694.509, Y 293.224, Z 438.017, A 0, B 90, C -64.379, E1 0, E2 0, E3 0, E4 0} C_DIS
LIN {X 694.212, Y 294.647, Z 437.848, A 0, B 90, C -64.44, E1 0, E2 0, E3 0, E4 0} C_DIS
LIN {X 693.909, Y 296.068, Z 437.674, A 0, B 90, C -64.501, E1 0, E2 0, E3 0, E4 0} C_DIS
LIN {X 693.599, Y 297.487, Z 437.497, A 0, B 90, C -64.563, E1 0, E2 0, E3 0, E4 0} C_DIS
LIN {X 693.282, Y 298.903, Z 437.315, A 0, B 90, C -64.624, E1 0, E2 0, E3 0, E4 0} C_DIS
LIN {X 692.958, Y 300.318, Z 437.13, A 0, B 90, C -64.686, E1 0, E2 0, E3 0, E4 0} C_DIS
LIN {X 692.628, Y 301.731, Z 436.941, A 0, B 90, C -64.749, E1 0, E2 0, E3 0, E4 0} C_DIS
LIN {X 692.291, Y 303.142, Z 436.749, A 0, B 90, C -64.811, E1 0, E2 0, E3 0, E4 0} C_DIS
LIN {X 691.948, Y 304.55, Z 436.552, A 0, B 90, C -64.873, E1 0, E2 0, E3 0, E4 0} C_DIS
LIN {X 691.598, Y 305.957, Z 436.352, A 0, B 90, C -64.936, E1 0, E2 0, E3 0, E4 0} C_DIS
LIN {X 691.241, Y 307.361, Z 436.147, A 0, B 90, C -64.999, E1 0, E2 0, E3 0, E4 0} C_DIS
LIN {X 690.877, Y 308.763, Z 435.939, A 0, B 90, C -65.062, E1 0, E2 0, E3 0, E4 0} C_DIS
LIN {X 690.507, Y 310.162, Z 435.728, A 0, B 90, C -65.125, E1 0, E2 0, E3 0, E4 0} C_DIS
LIN {X 690.13, Y 311.559, Z 435.512, A 0, B 90, C -65.189, E1 0, E2 0, E3 0, E4 0} C_DIS
LIN {X 689.747, Y 312.954, Z 435.293, A 0, B 90, C -65.252, E1 0, E2 0, E3 0, E4 0} C_DIS
LIN {X 689.357, Y 314.346, Z 435.07, A 0, B 90, C -65.316, E1 0, E2 0, E3 0, E4 0} C_DIS
LIN {X 688.96, Y 315.736, Z 434.843, A 0, B 90, C -65.38, E1 0, E2 0, E3 0, E4 0} C_DIS
LIN {X 688.557, Y 317.124, Z 434.612, A 0, B 90, C -65.444, E1 0, E2 0, E3 0, E4 0} C_DIS
LIN {X 688.147, Y 318.509, Z 434.377, A 0, B 90, C -65.508, E1 0, E2 0, E3 0, E4 0} C_DIS
LIN {X 687.731, Y 319.891, Z 434.139, A 0, B 90, C -65.572, E1 0, E2 0, E3 0, E4 0} C_DIS
LIN {X 687.308, Y 321.27, Z 433.897, A 0, B 90, C -65.637, E1 0, E2 0, E3 0, E4 0} C_DIS
LIN {X 686.879, Y 322.647, Z 433.652, A 0, B 90, C -65.702, E1 0, E2 0, E3 0, E4 0} C_DIS
LIN {X 686.443, Y 324.021, Z 433.402, A 0, B 90, C -65.767, E1 0, E2 0, E3 0, E4 0} C_DIS
LIN {X 686, Y 325.393, Z 433.149, A 0, B 90, C -65.832, E1 0, E2 0, E3 0, E4 0} C_DIS
LIN {X 685.551, Y 326.761, Z 432.892, A 0, B 90, C -65.897, E1 0, E2 0, E3 0, E4 0} C_DIS
LIN {X 685.096, Y 328.127, Z 432.632, A 0, B 90, C -65.962, E1 0, E2 0, E3 0, E4 0} C_DIS
LIN {X 684.634, Y 329.49, Z 432.367, A 0, B 90, C -66.028, E1 0, E2 0, E3 0, E4 0} C_DIS
LIN {X 684.166, Y 330.85, Z 432.099, A 0, B 90, C -66.094, E1 0, E2 0, E3 0, E4 0} C_DIS
LIN {X 683.691, Y 332.207, Z 431.828, A 0, B 90, C -66.159, E1 0, E2 0, E3 0, E4 0} C_DIS
LIN {X 683.21, Y 333.561, Z 431.553, A 0, B 90, C -66.225, E1 0, E2 0, E3 0, E4 0} C_DIS
LIN {X 682.722, Y 334.912, Z 431.274, A 0, B 90, C -66.292, E1 0, E2 0, E3 0, E4 0} C_DIS
LIN {X 682.229, Y 336.26, Z 430.991, A 0, B 90, C -66.358, E1 0, E2 0, E3 0, E4 0} C_DIS
LIN {X 681.728, Y 337.605, Z 430.705, A 0, B 90, C -66.424, E1 0, E2 0, E3 0, E4 0} C_DIS
LIN {X 681.221, Y 338.946, Z 430.415, A 0, B 90, C -66.491, E1 0, E2 0, E3 0, E4 0} C_DIS
LIN {X 680.708, Y 340.285, Z 430.121, A 0, B 90, C -66.558, E1 0, E2 0, E3 0, E4 0} C_DIS
LIN {X 680.189, Y 341.62, Z 429.824, A 0, B 90, C -66.624, E1 0, E2 0, E3 0, E4 0} C_DIS
LIN {X 679.663, Y 342.952, Z 429.523, A 0, B 90, C -66.691, E1 0, E2 0, E3 0, E4 0} C_DIS
LIN {X 679.131, Y 344.28, Z 429.219, A 0, B 90, C -66.759, E1 0, E2 0, E3 0, E4 0} C_DIS
LIN {X 678.593, Y 345.605, Z 428.911, A 0, B 90, C -66.826, E1 0, E2 0, E3 0, E4 0} C_DIS
LIN {X 678.049, Y 346.927, Z 428.599, A 0, B 90, C -66.893, E1 0, E2 0, E3 0, E4 0} C_DIS
LIN {X 677.498, Y 348.245, Z 428.284, A 0, B 90, C -66.961, E1 0, E2 0, E3 0, E4 0} C_DIS
LIN {X 676.941, Y 349.56, Z 427.965, A 0, B 90, C -67.028, E1 0, E2 0, E3 0, E4 0} C_DIS
LIN {X 676.377, Y 350.871, Z 427.643, A 0, B 90, C -67.096, E1 0, E2 0, E3 0, E4 0} C_DIS
LIN {X 675.808, Y 352.179, Z 427.317, A 0, B 90, C -67.164, E1 0, E2 0, E3 0, E4 0} C_DIS
LIN {X 675.232, Y 353.483, Z 426.988, A 0, B 90, C -67.232, E1 0, E2 0, E3 0, E4 0} C_DIS
LIN {X 674.65, Y 354.784, Z 426.655, A 0, B 90, C -67.3, E1 0, E2 0, E3 0, E4 0} C_DIS
LIN {X 674.063, Y 356.08, Z 426.318, A 0, B 90, C -67.369, E1 0, E2 0, E3 0, E4 0} C_DIS
LIN {X 673.468, Y 357.373, Z 425.979, A 0, B 90, C -67.437, E1 0, E2 0, E3 0, E4 0} C_DIS
LIN {X 672.868, Y 358.663, Z 425.635, A 0, B 90, C -67.506, E1 0, E2 0, E3 0, E4 0} C_DIS
LIN {X 672.262, Y 359.948, Z 425.288, A 0, B 90, C -67.575, E1 0, E2 0, E3 0, E4 0} C_DIS
LIN {X 671.649, Y 361.23, Z 424.938, A 0, B 90, C -67.643, E1 0, E2 0, E3 0, E4 0} C_DIS
LIN {X 671.031, Y 362.508, Z 424.584, A 0, B 90, C -67.712, E1 0, E2 0, E3 0, E4 0} C_DIS
LIN {X 670.406, Y 363.782, Z 424.227, A 0, B 90, C -67.781, E1 0, E2 0, E3 0, E4 0} C_DIS
LIN {X 669.776, Y 365.052, Z 423.866, A 0, B 90, C -67.851, E1 0, E2 0, E3 0, E4 0} C_DIS
LIN {X 669.139, Y 366.318, Z 423.501, A 0, B 90, C -67.92, E1 0, E2 0, E3 0, E4 0} C_DIS
LIN {X 668.497, Y 367.58, Z 423.134, A 0, B 90, C -67.989, E1 0, E2 0, E3 0, E4 0} C_DIS
LIN {X 667.848, Y 368.838, Z 422.763, A 0, B 90, C -68.059, E1 0, E2 0, E3 0, E4 0} C_DIS
LIN {X 667.194, Y 370.091, Z 422.388, A 0, B 90, C -68.128, E1 0, E2 0, E3 0, E4 0} C_DIS
LIN {X 666.533, Y 371.341, Z 422.01, A 0, B 90, C -68.198, E1 0, E2 0, E3 0, E4 0} C_DIS
LIN {X 665.867, Y 372.587, Z 421.629, A 0, B 90, C -68.268, E1 0, E2 0, E3 0, E4 0} C_DIS
LIN {X 665.195, Y 373.828, Z 421.245, A 0, B 90, C -68.338, E1 0, E2 0, E3 0, E4 0} C_DIS
LIN {X 664.517, Y 375.065, Z 420.857, A 0, B 90, C -68.408, E1 0, E2 0, E3 0, E4 0} C_DIS
LIN {X 663.833, Y 376.298, Z 420.465, A 0, B 90, C -68.478, E1 0, E2 0, E3 0, E4 0} C_DIS
LIN {X 663.143, Y 377.526, Z 420.071, A 0, B 90, C -68.549, E1 0, E2 0, E3 0, E4 0} C_DIS
LIN {X 662.447, Y 378.75, Z 419.673, A 0, B 90, C -68.619, E1 0, E2 0, E3 0, E4 0} C_DIS
LIN {X 661.746, Y 379.97, Z 419.271, A 0, B 90, C -68.69, E1 0, E2 0, E3 0, E4 0} C_DIS
LIN {X 661.039, Y 381.185, Z 418.867, A 0, B 90, C -68.76, E1 0, E2 0, E3 0, E4 0} C_DIS
LIN {X 660.326, Y 382.396, Z 418.459, A 0, B 90, C -68.831, E1 0, E2 0, E3 0, E4 0} C_DIS
LIN {X 659.607, Y 383.602, Z 418.048, A 0, B 90, C -68.902, E1 0, E2 0, E3 0, E4 0} C_DIS
LIN {X 658.883, Y 384.804, Z 417.633, A 0, B 90, C -68.973, E1 0, E2 0, E3 0, E4 0} C_DIS
LIN {X 658.153, Y 386.001, Z 417.216, A 0, B 90, C -69.044, E1 0, E2 0, E3 0, E4 0} C_DIS
LIN {X 657.417, Y 387.194, Z 416.795, A 0, B 90, C -69.115, E1 0, E2 0, E3 0, E4 0} C_DIS
LIN {X 656.676, Y 388.382, Z 416.37, A 0, B 90, C -69.186, E1 0, E2 0, E3 0, E4 0} C_DIS
LIN {X 655.929, Y 389.565, Z 415.943, A 0, B 90, C -69.257, E1 0, E2 0, E3 0, E4 0} C_DIS
LIN {X 655.177, Y 390.744, Z 415.513, A 0, B 90, C -69.329, E1 0, E2 0, E3 0, E4 0} C_DIS
LIN {X 654.419, Y 391.917, Z 415.079, A 0, B 90, C -69.4, E1 0, E2 0, E3 0, E4 0} C_DIS
LIN {X 653.655, Y 393.086, Z 414.642, A 0, B 90, C -69.472, E1 0, E2 0, E3 0, E4 0} C_DIS
LIN {X 652.886, Y 394.251, Z 414.202, A 0, B 90, C -69.543, E1 0, E2 0, E3 0, E4 0} C_DIS
LIN {X 652.111, Y 395.41, Z 413.759, A 0, B 90, C -69.615, E1 0, E2 0, E3 0, E4 0} C_DIS
LIN {X 651.331, Y 396.564, Z 413.312, A 0, B 90, C -69.687, E1 0, E2 0, E3 0, E4 0} C_DIS
LIN {X 650.545, Y 397.714, Z 412.863, A 0, B 90, C -69.759, E1 0, E2 0, E3 0, E4 0} C_DIS
LIN {X 649.754, Y 398.858, Z 412.41, A 0, B 90, C -69.831, E1 0, E2 0, E3 0, E4 0} C_DIS
LIN {X 648.958, Y 399.998, Z 411.954, A 0, B 90, C -69.903, E1 0, E2 0, E3 0, E4 0} C_DIS
LIN {X 648.156, Y 401.132, Z 411.496, A 0, B 90, C -69.975, E1 0, E2 0, E3 0, E4 0} C_DIS
LIN {X 647.349, Y 402.262, Z 411.034, A 0, B 90, C -70.048, E1 0, E2 0, E3 0, E4 0} C_DIS
LIN {X 646.536, Y 403.386, Z 410.569, A 0, B 90, C -70.12, E1 0, E2 0, E3 0, E4 0} C_DIS
LIN {X 645.719, Y 404.506, Z 410.101, A 0, B 90, C -70.192, E1 0, E2 0, E3 0, E4 0} C_DIS
LIN {X 644.895, Y 405.62, Z 409.63, A 0, B 90, C -70.265, E1 0, E2 0, E3 0, E4 0} C_DIS
LIN {X 644.067, Y 406.729, Z 409.156, A 0, B 90, C -70.338, E1 0, E2 0, E3 0, E4 0} C_DIS
LIN {X 643.233, Y 407.832, Z 408.679, A 0, B 90, C -70.41, E1 0, E2 0, E3 0, E4 0} C_DIS
LIN {X 642.394, Y 408.931, Z 408.199, A 0, B 90, C -70.483, E1 0, E2 0, E3 0, E4 0} C_DIS
LIN {X 641.55, Y 410.024, Z 407.716, A 0, B 90, C -70.556, E1 0, E2 0, E3 0, E4 0} C_DIS
LIN {X 640.701, Y 411.112, Z 407.23, A 0, B 90, C -70.629, E1 0, E2 0, E3 0, E4 0} C_DIS
LIN {X 639.847, Y 412.194, Z 406.741, A 0, B 90, C -70.702, E1 0, E2 0, E3 0, E4 0} C_DIS
LIN {X 638.987, Y 413.271, Z 406.249, A 0, B 90, C -70.775, E1 0, E2 0, E3 0, E4 0} C_DIS
LIN {X 638.123, Y 414.343, Z 405.755, A 0, B 90, C -70.848, E1 0, E2 0, E3 0, E4 0} C_DIS
LIN {X 637.253, Y 415.409, Z 405.257, A 0, B 90, C -70.921, E1 0, E2 0, E3 0, E4 0} C_DIS
LIN {X 636.378, Y 416.47, Z 404.757, A 0, B 90, C -70.994, E1 0, E2 0, E3 0, E4 0} C_DIS
LIN {X 635.499, Y 417.525, Z 404.253, A 0, B 90, C -71.068, E1 0, E2 0, E3 0, E4 0} C_DIS
LIN {X 634.614, Y 418.574, Z 403.747, A 0, B 90, C -71.141, E1 0, E2 0, E3 0, E4 0} C_DIS
LIN {X 633.724, Y 419.618, Z 403.238, A 0, B 90, C -71.215, E1 0, E2 0, E3 0, E4 0} C_DIS
LIN {X 632.83, Y 420.657, Z 402.726, A 0, B 90, C -71.288, E1 0, E2 0, E3 0, E4 0} C_DIS
LIN {X 631.93, Y 421.69, Z 402.212, A 0, B 90, C -71.362, E1 0, E2 0, E3 0, E4 0} C_DIS
LIN {X 631.026, Y 422.717, Z 401.694, A 0, B 90, C -71.435, E1 0, E2 0, E3 0, E4 0} C_DIS
LIN {X 630.117, Y 423.738, Z 401.174, A 0, B 90, C -71.509, E1 0, E2 0, E3 0, E4 0} C_DIS
LIN {X 629.203, Y 424.754, Z 400.651, A 0, B 90, C -71.583, E1 0, E2 0, E3 0, E4 0} C_DIS
LIN {X 628.284, Y 425.764, Z 400.125, A 0, B 90, C -71.657, E1 0, E2 0, E3 0, E4 0} C_DIS
LIN {X 627.36, Y 426.768, Z 399.597, A 0, B 90, C -71.731, E1 0, E2 0, E3 0, E4 0} C_DIS
LIN {X 626.432, Y 427.766, Z 399.066, A 0, B 90, C -71.805, E1 0, E2 0, E3 0, E4 0} C_DIS
LIN {X 625.499, Y 428.759, Z 398.532, A 0, B 90, C -71.879, E1 0, E2 0, E3 0, E4 0} C_DIS
LIN {X 624.561, Y 429.745, Z 397.995, A 0, B 90, C -71.953, E1 0, E2 0, E3 0, E4 0} C_DIS
LIN {X 623.619, Y 430.726, Z 397.456, A 0, B 90, C -72.027, E1 0, E2 0, E3 0, E4 0} C_DIS
LIN {X 622.672, Y 431.701, Z 396.914, A 0, B 90, C -72.101, E1 0, E2 0, E3 0, E4 0} C_DIS
LIN {X 621.72, Y 432.669, Z 396.369, A 0, B 90, C -72.175, E1 0, E2 0, E3 0, E4 0} C_DIS
LIN {X 620.764, Y 433.632, Z 395.822, A 0, B 90, C -72.25, E1 0, E2 0, E3 0, E4 0} C_DIS
LIN {X 619.803, Y 434.589, Z 395.273, A 0, B 90, C -72.324, E1 0, E2 0, E3 0, E4 0} C_DIS
LIN {X 618.838, Y 435.54, Z 394.72, A 0, B 90, C -72.399, E1 0, E2 0, E3 0, E4 0} C_DIS
LIN {X 617.868, Y 436.484, Z 394.165, A 0, B 90, C -72.473, E1 0, E2 0, E3 0, E4 0} C_DIS
LIN {X 616.894, Y 437.423, Z 393.608, A 0, B 90, C -72.548, E1 0, E2 0, E3 0, E4 0} C_DIS
LIN {X 615.915, Y 438.355, Z 393.048, A 0, B 90, C -72.622, E1 0, E2 0, E3 0, E4 0} C_DIS
LIN {X 614.932, Y 439.281, Z 392.485, A 0, B 90, C -72.697, E1 0, E2 0, E3 0, E4 0} C_DIS
LIN {X 613.944, Y 440.201, Z 391.92, A 0, B 90, C -72.772, E1 0, E2 0, E3 0, E4 0} C_DIS
LIN {X 612.953, Y 441.115, Z 391.353, A 0, B 90, C -72.846, E1 0, E2 0, E3 0, E4 0} C_DIS
LIN {X 611.957, Y 442.022, Z 390.783, A 0, B 90, C -72.921, E1 0, E2 0, E3 0, E4 0} C_DIS
LIN {X 610.956, Y 442.923, Z 390.211, A 0, B 90, C -72.996, E1 0, E2 0, E3 0, E4 0} C_DIS
LIN {X 609.951, Y 443.818, Z 389.636, A 0, B 90, C -73.071, E1 0, E2 0, E3 0, E4 0} C_DIS
LIN {X 608.943, Y 444.707, Z 389.059, A 0, B 90, C -73.146, E1 0, E2 0, E3 0, E4 0} C_DIS
LIN {X 607.93, Y 445.589, Z 388.479, A 0, B 90, C -73.221, E1 0, E2 0, E3 0, E4 0} C_DIS
LIN {X 606.912, Y 446.465, Z 387.897, A 0, B 90, C -73.296, E1 0, E2 0, E3 0, E4 0} C_DIS
LIN {X 605.891, Y 447.334, Z 387.312, A 0, B 90, C -73.371, E1 0, E2 0, E3 0, E4 0} C_DIS
LIN {X 604.865, Y 448.197, Z 386.726, A 0, B 90, C -73.446, E1 0, E2 0, E3 0, E4 0} C_DIS
LIN {X 603.836, Y 449.054, Z 386.137, A 0, B 90, C -73.521, E1 0, E2 0, E3 0, E4 0} C_DIS
LIN {X 602.802, Y 449.904, Z 385.545, A 0, B 90, C -73.596, E1 0, E2 0, E3 0, E4 0} C_DIS
LIN {X 601.765, Y 450.747, Z 384.952, A 0, B 90, C -73.671, E1 0, E2 0, E3 0, E4 0} C_DIS
LIN {X 600.723, Y 451.584, Z 384.356, A 0, B 90, C -73.747, E1 0, E2 0, E3 0, E4 0} C_DIS
LIN {X 599.678, Y 452.415, Z 383.757, A 0, B 90, C -73.822, E1 0, E2 0, E3 0, E4 0} C_DIS
LIN {X 598.628, Y 453.239, Z 383.157, A 0, B 90, C -73.897, E1 0, E2 0, E3 0, E4 0} C_DIS
LIN {X 597.575, Y 454.056, Z 382.554, A 0, B 90, C -73.973, E1 0, E2 0, E3 0, E4 0} C_DIS
LIN {X 596.518, Y 454.866, Z 381.949, A 0, B 90, C -74.048, E1 0, E2 0, E3 0, E4 0} C_DIS
LIN {X 595.457, Y 455.67, Z 381.342, A 0, B 90, C -74.123, E1 0, E2 0, E3 0, E4 0} C_DIS
LIN {X 594.392, Y 456.467, Z 380.733, A 0, B 90, C -74.199, E1 0, E2 0, E3 0, E4 0} C_DIS
LIN {X 593.323, Y 457.258, Z 380.121, A 0, B 90, C -74.274, E1 0, E2 0, E3 0, E4 0} C_DIS
LIN {X 592.251, Y 458.042, Z 379.508, A 0, B 90, C -74.35, E1 0, E2 0, E3 0, E4 0} C_DIS
LIN {X 591.175, Y 458.819, Z 378.892, A 0, B 90, C -74.426, E1 0, E2 0, E3 0, E4 0} C_DIS
LIN {X 590.095, Y 459.589, Z 378.275, A 0, B 90, C -74.501, E1 0, E2 0, E3 0, E4 0} C_DIS
LIN {X 589.012, Y 460.353, Z 377.655, A 0, B 90, C -74.577, E1 0, E2 0, E3 0, E4 0} C_DIS
LIN {X 587.925, Y 461.109, Z 377.033, A 0, B 90, C -74.652, E1 0, E2 0, E3 0, E4 0} C_DIS
LIN {X 586.834, Y 461.859, Z 376.409, A 0, B 90, C -74.728, E1 0, E2 0, E3 0, E4 0} C_DIS
LIN {X 585.74, Y 462.602, Z 375.783, A 0, B 90, C -74.804, E1 0, E2 0, E3 0, E4 0} C_DIS
LIN {X 584.643, Y 463.338, Z 375.155, A 0, B 90, C -74.88, E1 0, E2 0, E3 0, E4 0} C_DIS
LIN {X 583.542, Y 464.067, Z 374.525, A 0, B 90, C -74.955, E1 0, E2 0, E3 0, E4 0} C_DIS
LIN {X 582.438, Y 464.789, Z 373.893, A 0, B 90, C -75.031, E1 0, E2 0, E3 0, E4 0} C_DIS
LIN {X 581.33, Y 465.504, Z 373.259, A 0, B 90, C -75.107, E1 0, E2 0, E3 0, E4 0} C_DIS
LIN {X 580.219, Y 466.213, Z 372.623, A 0, B 90, C -75.183, E1 0, E2 0, E3 0, E4 0} C_DIS
LIN {X 579.104, Y 466.914, Z 371.986, A 0, B 90, C -75.259, E1 0, E2 0, E3 0, E4 0} C_DIS
LIN {X 577.986, Y 467.608, Z 371.346, A 0, B 90, C -75.335, E1 0, E2 0, E3 0, E4 0} C_DIS
LIN {X 576.865, Y 468.295, Z 370.705, A 0, B 90, C -75.41, E1 0, E2 0, E3 0, E4 0} C_DIS
LIN {X 575.741, Y 468.975, Z 370.061, A 0, B 90, C -75.486, E1 0, E2 0, E3 0, E4 0} C_DIS
LIN {X 574.613, Y 469.648, Z 369.416, A 0, B 90, C -75.562, E1 0, E2 0, E3 0, E4 0} C_DIS
LIN {X 573.482, Y 470.314, Z 368.769, A 0, B 90, C -75.638, E1 0, E2 0, E3 0, E4 0} C_DIS
LIN {X 572.348, Y 470.973, Z 368.12, A 0, B 90, C -75.714, E1 0, E2 0, E3 0, E4 0} C_DIS
LIN {X 571.211, Y 471.625, Z 367.47, A 0, B 90, C -75.79, E1 0, E2 0, E3 0, E4 0} C_DIS
LIN {X 570.071, Y 472.269, Z 366.817, A 0, B 90, C -75.866, E1 0, E2 0, E3 0, E4 0} C_DIS
LIN {X 568.928, Y 472.907, Z 366.163, A 0, B 90, C -75.942, E1 0, E2 0, E3 0, E4 0} C_DIS
LIN {X 567.782, Y 473.537, Z 365.508, A 0, B 90, C -76.018, E1 0, E2 0, E3 0, E4 0} C_DIS
LIN {X 566.633, Y 474.16, Z 364.85, A 0, B 90, C -76.094, E1 0, E2 0, E3 0, E4 0} C_DIS
LIN {X 565.481, Y 474.775, Z 364.191, A 0, B 90, C -76.171, E1 0, E2 0, E3 0, E4 0} C_DIS
LIN {X 564.326, Y 475.384, Z 363.53, A 0, B 90, C -76.247, E1 0, E2 0, E3 0, E4 0} C_DIS
LIN {X 563.168, Y 475.985, Z 362.868, A 0, B 90, C -76.323, E1 0, E2 0, E3 0, E4 0} C_DIS
LIN {X 562.008, Y 476.579, Z 362.204, A 0, B 90, C -76.399, E1 0, E2 0, E3 0, E4 0} C_DIS
LIN {X 560.845, Y 477.165, Z 361.538, A 0, B 90, C -76.475, E1 0, E2 0, E3 0, E4 0} C_DIS
LIN {X 559.678, Y 477.744, Z 360.871, A 0, B 90, C -76.551, E1 0, E2 0, E3 0, E4 0} C_DIS
LIN {X 558.51, Y 478.316, Z 360.202, A 0, B 90, C -76.627, E1 0, E2 0, E3 0, E4 0} C_DIS
LIN {X 557.338, Y 478.881, Z 359.532, A 0, B 90, C -76.704, E1 0, E2 0, E3 0, E4 0} C_DIS
LIN {X 556.164, Y 479.438, Z 358.86, A 0, B 90, C -76.78, E1 0, E2 0, E3 0, E4 0} C_DIS
LIN {X 554.987, Y 479.988, Z 358.186, A 0, B 90, C -76.856, E1 0, E2 0, E3 0, E4 0} C_DIS
LIN {X 553.807, Y 480.53, Z 357.512, A 0, B 90, C -76.932, E1 0, E2 0, E3 0, E4 0} C_DIS
LIN {X 552.625, Y 481.065, Z 356.835, A 0, B 90, C -77.008, E1 0, E2 0, E3 0, E4 0} C_DIS
LIN {X 551.441, Y 481.592, Z 356.158, A 0, B 90, C -77.085, E1 0, E2 0, E3 0, E4 0} C_DIS
LIN {X 550.254, Y 482.112, Z 355.478, A 0, B 90, C -77.161, E1 0, E2 0, E3 0, E4 0} C_DIS
LIN {X 549.065, Y 482.625, Z 354.798, A 0, B 90, C -77.237, E1 0, E2 0, E3 0, E4 0} C_DIS
LIN {X 547.873, Y 483.13, Z 354.116, A 0, B 90, C -77.313, E1 0, E2 0, E3 0, E4 0} C_DIS
LIN {X 546.678, Y 483.628, Z 353.433, A 0, B 90, C -77.389, E1 0, E2 0, E3 0, E4 0} C_DIS
LIN {X 545.482, Y 484.118, Z 352.748, A 0, B 90, C -77.466, E1 0, E2 0, E3 0, E4 0} C_DIS
LIN {X 544.283, Y 484.6, Z 352.062, A 0, B 90, C -77.542, E1 0, E2 0, E3 0, E4 0} C_DIS
LIN {X 543.082, Y 485.075, Z 351.375, A 0, B 90, C -77.618, E1 0, E2 0, E3 0, E4 0} C_DIS
LIN {X 541.879, Y 485.542, Z 350.686, A 0, B 90, C -77.694, E1 0, E2 0, E3 0, E4 0} C_DIS
LIN {X 540.673, Y 486.002, Z 349.996, A 0, B 90, C -77.771, E1 0, E2 0, E3 0, E4 0} C_DIS
LIN {X 539.465, Y 486.454, Z 349.305, A 0, B 90, C -77.847, E1 0, E2 0, E3 0, E4 0} C_DIS
LIN {X 538.255, Y 486.899, Z 348.613, A 0, B 90, C -77.923, E1 0, E2 0, E3 0, E4 0} C_DIS
LIN {X 537.044, Y 487.336, Z 347.92, A 0, B 90, C -77.999, E1 0, E2 0, E3 0, E4 0} C_DIS
LIN {X 535.83, Y 487.765, Z 347.225, A 0, B 90, C -78.076, E1 0, E2 0, E3 0, E4 0} C_DIS
LIN {X 534.614, Y 488.187, Z 346.529, A 0, B 90, C -78.152, E1 0, E2 0, E3 0, E4 0} C_DIS
LIN {X 533.396, Y 488.601, Z 345.832, A 0, B 90, C -78.228, E1 0, E2 0, E3 0, E4 0} C_DIS
LIN {X 532.176, Y 489.008, Z 345.134, A 0, B 90, C -78.304, E1 0, E2 0, E3 0, E4 0} C_DIS
LIN {X 530.954, Y 489.406, Z 344.435, A 0, B 90, C -78.381, E1 0, E2 0, E3 0, E4 0} C_DIS
LIN {X 529.73, Y 489.797, Z 343.735, A 0, B 90, C -78.457, E1 0, E2 0, E3 0, E4 0} C_DIS
LIN {X 528.505, Y 490.181, Z 343.034, A 0, B 90, C -78.533, E1 0, E2 0, E3 0, E4 0} C_DIS
LIN {X 527.277, Y 490.556, Z 342.332, A 0, B 90, C -78.609, E1 0, E2 0, E3 0, E4 0} C_DIS
LIN {X 526.048, Y 490.924, Z 341.628, A 0, B 90, C -78.685, E1 0, E2 0, E3 0, E4 0} C_DIS
LIN {X 524.817, Y 491.285, Z 340.924, A 0, B 90, C -78.762, E1 0, E2 0, E3 0, E4 0} C_DIS
LIN {X 523.585, Y 491.637, Z 340.219, A 0, B 90, C -78.838, E1 0, E2 0, E3 0, E4 0} C_DIS
LIN {X 522.351, Y 491.982, Z 339.513, A 0, B 90, C -78.914, E1 0, E2 0, E3 0, E4 0} C_DIS
LIN {X 521.115, Y 492.319, Z 338.806, A 0, B 90, C -78.99, E1 0, E2 0, E3 0, E4 0} C_DIS
LIN {X 519.878, Y 492.648, Z 338.098, A 0, B 90, C -79.066, E1 0, E2 0, E3 0, E4 0} C_DIS
LIN {X 518.639, Y 492.969, Z 337.389, A 0, B 90, C -79.142, E1 0, E2 0, E3 0, E4 0} C_DIS
LIN {X 517.398, Y 493.283, Z 336.679, A 0, B 90, C -79.218, E1 0, E2 0, E3 0, E4 0} C_DIS
LIN {X 516.156, Y 493.588, Z 335.969, A 0, B 90, C -79.295, E1 0, E2 0, E3 0, E4 0} C_DIS
LIN {X 514.913, Y 493.886, Z 335.257, A 0, B 90, C -79.371, E1 0, E2 0, E3 0, E4 0} C_DIS
LIN {X 513.668, Y 494.176, Z 334.545, A 0, B 90, C -79.447, E1 0, E2 0, E3 0, E4 0} C_DIS
LIN {X 512.422, Y 494.459, Z 333.832, A 0, B 90, C -79.523, E1 0, E2 0, E3 0, E4 0} C_DIS
LIN {X 511.175, Y 494.733, Z 333.118, A 0, B 90, C -79.599, E1 0, E2 0, E3 0, E4 0} C_DIS
LIN {X 509.926, Y 495, Z 332.404, A 0, B 90, C -79.675, E1 0, E2 0, E3 0, E4 0} C_DIS
LIN {X 508.676, Y 495.258, Z 331.689, A 0, B 90, C -79.751, E1 0, E2 0, E3 0, E4 0} C_DIS
LIN {X 507.425, Y 495.509, Z 330.973, A 0, B 90, C -79.827, E1 0, E2 0, E3 0, E4 0} C_DIS
LIN {X 506.173, Y 495.752, Z 330.256, A 0, B 90, C -79.903, E1 0, E2 0, E3 0, E4 0} C_DIS
LIN {X 504.92, Y 495.987, Z 329.539, A 0, B 90, C -79.979, E1 0, E2 0, E3 0, E4 0} C_DIS
LIN {X 503.665, Y 496.214, Z 328.821, A 0, B 90, C -80.055, E1 0, E2 0, E3 0, E4 0} C_DIS
LIN {X 502.41, Y 496.434, Z 328.103, A 0, B 90, C -80.131, E1 0, E2 0, E3 0, E4 0} C_DIS
LIN {X 501.153, Y 496.645, Z 327.384, A 0, B 90, C -80.207, E1 0, E2 0, E3 0, E4 0} C_DIS
LIN {X 499.896, Y 496.849, Z 326.665, A 0, B 90, C -80.283, E1 0, E2 0, E3 0, E4 0} C_DIS
LIN {X 498.637, Y 497.044, Z 325.944, A 0, B 90, C -80.359, E1 0, E2 0, E3 0, E4 0} C_DIS
LIN {X 497.378, Y 497.232, Z 325.224, A 0, B 90, C -80.434, E1 0, E2 0, E3 0, E4 0} C_DIS
LIN {X 496.117, Y 497.412, Z 324.503, A 0, B 90, C -80.51, E1 0, E2 0, E3 0, E4 0} C_DIS
LIN {X 494.856, Y 497.584, Z 323.781, A 0, B 90, C -80.586, E1 0, E2 0, E3 0, E4 0} C_DIS
LIN {X 493.594, Y 497.747, Z 323.059, A 0, B 90, C -80.662, E1 0, E2 0, E3 0, E4 0} C_DIS
LIN {X 492.332, Y 497.903, Z 322.337, A 0, B 90, C -80.738, E1 0, E2 0, E3 0, E4 0} C_DIS
LIN {X 491.068, Y 498.051, Z 321.614, A 0, B 90, C -80.813, E1 0, E2 0, E3 0, E4 0} C_DIS
LIN {X 489.804, Y 498.191, Z 320.891, A 0, B 90, C -80.889, E1 0, E2 0, E3 0, E4 0} C_DIS
LIN {X 488.539, Y 498.324, Z 320.167, A 0, B 90, C -80.965, E1 0, E2 0, E3 0, E4 0} C_DIS
LIN {X 487.274, Y 498.448, Z 319.443, A 0, B 90, C -81.04, E1 0, E2 0, E3 0, E4 0} C_DIS
LIN {X 486.008, Y 498.564, Z 318.719, A 0, B 90, C -81.116, E1 0, E2 0, E3 0, E4 0} C_DIS
LIN {X 484.742, Y 498.672, Z 317.994, A 0, B 90, C -81.192, E1 0, E2 0, E3 0, E4 0} C_DIS
LIN {X 483.475, Y 498.772, Z 317.269, A 0, B 90, C -81.267, E1 0, E2 0, E3 0, E4 0} C_DIS
LIN {X 482.208, Y 498.865, Z 316.544, A 0, B 90, C -81.343, E1 0, E2 0, E3 0, E4 0} C_DIS
LIN {X 480.94, Y 498.949, Z 315.819, A 0, B 90, C -81.418, E1 0, E2 0, E3 0, E4 0} C_DIS
LIN {X 479.672, Y 499.025, Z 315.093, A 0, B 90, C -81.494, E1 0, E2 0, E3 0, E4 0} C_DIS
LIN {X 478.403, Y 499.094, Z 314.367, A 0, B 90, C -81.569, E1 0, E2 0, E3 0, E4 0} C_DIS
LIN {X 477.134, Y 499.154, Z 313.641, A 0, B 90, C -81.644, E1 0, E2 0, E3 0, E4 0} C_DIS
LIN {X 475.865, Y 499.207, Z 312.915, A 0, B 90, C -81.72, E1 0, E2 0, E3 0, E4 0} C_DIS
LIN {X 474.596, Y 499.251, Z 312.189, A 0, B 90, C -81.795, E1 0, E2 0, E3 0, E4 0} C_DIS
LIN {X 473.326, Y 499.287, Z 311.462, A 0, B 90, C -81.87, E1 0, E2 0, E3 0, E4 0} C_DIS
LIN {X 472.057, Y 499.316, Z 310.736, A 0, B 90, C -81.946, E1 0, E2 0, E3 0, E4 0} C_DIS
LIN {X 470.787, Y 499.336, Z 310.009, A 0, B 90, C -82.021, E1 0, E2 0, E3 0, E4 0} C_DIS
LIN {X 469.517, Y 499.349, Z 309.283, A 0, B 90, C -82.096, E1 0, E2 0, E3 0, E4 0} C_DIS
LIN {X 468.247, Y 499.353, Z 308.556, A 0, B 90, C -82.171, E1 0, E2 0, E3 0, E4 0} C_DIS
LIN {X 466.977, Y 499.35, Z 307.83, A 0, B 90, C -82.246, E1 0, E2 0, E3 0, E4 0} C_DIS
LIN {X 465.707, Y 499.338, Z 307.103, A 0, B 90, C -82.322, E1 0, E2 0, E3 0, E4 0} C_DIS
LIN {X 464.438, Y 499.319, Z 306.376, A 0, B 90, C -82.397, E1 0, E2 0, E3 0, E4 0} C_DIS
LIN {X 463.168, Y 499.292, Z 305.65, A 0, B 90, C -82.472, E1 0, E2 0, E3 0, E4 0} C_DIS
LIN {X 461.898, Y 499.256, Z 304.924, A 0, B 90, C -82.547, E1 0, E2 0, E3 0, E4 0} C_DIS
LIN {X 460.629, Y 499.213, Z 304.197, A 0, B 90, C -82.621, E1 0, E2 0, E3 0, E4 0} C_DIS
LIN {X 459.36, Y 499.161, Z 303.471, A 0, B 90, C -82.696, E1 0, E2 0, E3 0, E4 0} C_DIS
LIN {X 458.091, Y 499.102, Z 302.745, A 0, B 90, C -82.771, E1 0, E2 0, E3 0, E4 0} C_DIS
LIN {X 456.823, Y 499.035, Z 302.019, A 0, B 90, C -82.846, E1 0, E2 0, E3 0, E4 0} C_DIS
LIN {X 455.554, Y 498.959, Z 301.294, A 0, B 90, C -82.921, E1 0, E2 0, E3 0, E4 0} C_DIS
LIN {X 454.286, Y 498.876, Z 300.568, A 0, B 90, C -82.995, E1 0, E2 0, E3 0, E4 0} C_DIS
LIN {X 453.019, Y 498.785, Z 299.843, A 0, B 90, C -83.07, E1 0, E2 0, E3 0, E4 0} C_DIS
LIN {X 451.752, Y 498.685, Z 299.118, A 0, B 90, C -83.145, E1 0, E2 0, E3 0, E4 0} C_DIS
LIN {X 450.486, Y 498.578, Z 298.393, A 0, B 90, C -83.219, E1 0, E2 0, E3 0, E4 0} C_DIS
LIN {X 449.22, Y 498.463, Z 297.669, A 0, B 90, C -83.294, E1 0, E2 0, E3 0, E4 0} C_DIS
LIN {X 447.954, Y 498.34, Z 296.945, A 0, B 90, C -83.368, E1 0, E2 0, E3 0, E4 0} C_DIS
LIN {X 446.689, Y 498.209, Z 296.221, A 0, B 90, C -83.443, E1 0, E2 0, E3 0, E4 0} C_DIS
LIN {X 445.425, Y 498.07, Z 295.498, A 0, B 90, C -83.517, E1 0, E2 0, E3 0, E4 0} C_DIS
LIN {X 444.162, Y 497.923, Z 294.775, A 0, B 90, C -83.591, E1 0, E2 0, E3 0, E4 0} C_DIS
LIN {X 442.899, Y 497.768, Z 294.053, A 0, B 90, C -83.666, E1 0, E2 0, E3 0, E4 0} C_DIS
LIN {X 441.637, Y 497.605, Z 293.331, A 0, B 90, C -83.74, E1 0, E2 0, E3 0, E4 0} C_DIS
LIN {X 440.376, Y 497.434, Z 292.609, A 0, B 90, C -83.814, E1 0, E2 0, E3 0, E4 0} C_DIS
LIN {X 439.115, Y 497.255, Z 291.888, A 0, B 90, C -83.888, E1 0, E2 0, E3 0, E4 0} C_DIS
LIN {X 437.856, Y 497.069, Z 291.167, A 0, B 90, C -83.962, E1 0, E2 0, E3 0, E4 0} C_DIS
LIN {X 436.597, Y 496.874, Z 290.447, A 0, B 90, C -84.036, E1 0, E2 0, E3 0, E4 0} C_DIS
LIN {X 435.34, Y 496.672, Z 289.727, A 0, B 90, C -84.11, E1 0, E2 0, E3 0, E4 0} C_DIS
LIN {X 434.083, Y 496.461, Z 289.008, A 0, B 90, C -84.184, E1 0, E2 0, E3 0, E4 0} C_DIS
LIN {X 432.827, Y 496.243, Z 288.29, A 0, B 90, C -84.258, E1 0, E2 0, E3 0, E4 0} C_DIS
LIN {X 431.573, Y 496.017, Z 287.572, A 0, B 90, C -84.332, E1 0, E2 0, E3 0, E4 0} C_DIS
LIN {X 430.319, Y 495.783, Z 286.855, A 0, B 90, C -84.406, E1 0, E2 0, E3 0, E4 0} C_DIS
LIN {X 429.067, Y 495.541, Z 286.138, A 0, B 90, C -84.479, E1 0, E2 0, E3 0, E4 0} C_DIS
LIN {X 427.815, Y 495.291, Z 285.422, A 0, B 90, C -84.553, E1 0, E2 0, E3 0, E4 0} C_DIS
LIN {X 426.565, Y 495.033, Z 284.707, A 0, B 90, C -84.626, E1 0, E2 0, E3 0, E4 0} C_DIS
LIN {X 425.317, Y 494.768, Z 283.992, A 0, B 90, C -84.7, E1 0, E2 0, E3 0, E4 0} C_DIS
LIN {X 424.069, Y 494.494, Z 283.279, A 0, B 90, C -84.773, E1 0, E2 0, E3 0, E4 0} C_DIS
LIN {X 422.823, Y 494.213, Z 282.565, A 0, B 90, C -84.847, E1 0, E2 0, E3 0, E4 0} C_DIS
LIN {X 421.578, Y 493.924, Z 281.853, A 0, B 90, C -84.92, E1 0, E2 0, E3 0, E4 0} C_DIS
LIN {X 420.334, Y 493.627, Z 281.142, A 0, B 90, C -84.993, E1 0, E2 0, E3 0, E4 0} C_DIS
LIN {X 419.092, Y 493.322, Z 280.431, A 0, B 90, C -85.066, E1 0, E2 0, E3 0, E4 0} C_DIS
LIN {X 417.852, Y 493.01, Z 279.721, A 0, B 90, C -85.14, E1 0, E2 0, E3 0, E4 0} C_DIS
LIN {X 416.613, Y 492.689, Z 279.012, A 0, B 90, C -85.213, E1 0, E2 0, E3 0, E4 0} C_DIS
LIN {X 415.375, Y 492.361, Z 278.304, A 0, B 90, C -85.286, E1 0, E2 0, E3 0, E4 0} C_DIS
LIN {X 414.139, Y 492.025, Z 277.597, A 0, B 90, C -85.359, E1 0, E2 0, E3 0, E4 0} C_DIS
LIN {X 412.905, Y 491.682, Z 276.891, A 0, B 90, C -85.431, E1 0, E2 0, E3 0, E4 0} C_DIS
LIN {X 411.672, Y 491.33, Z 276.185, A 0, B 90, C -85.504, E1 0, E2 0, E3 0, E4 0} C_DIS
LIN {X 410.441, Y 490.971, Z 275.481, A 0, B 90, C -85.577, E1 0, E2 0, E3 0, E4 0} C_DIS
LIN {X 409.212, Y 490.604, Z 274.778, A 0, B 90, C -85.65, E1 0, E2 0, E3 0, E4 0} C_DIS
LIN {X 407.984, Y 490.229, Z 274.075, A 0, B 90, C -85.722, E1 0, E2 0, E3 0, E4 0} C_DIS
LIN {X 406.758, Y 489.847, Z 273.374, A 0, B 90, C -85.795, E1 0, E2 0, E3 0, E4 0} C_DIS
LIN {X 405.534, Y 489.457, Z 272.674, A 0, B 90, C -85.867, E1 0, E2 0, E3 0, E4 0} C_DIS
LIN {X 404.312, Y 489.059, Z 271.974, A 0, B 90, C -85.939, E1 0, E2 0, E3 0, E4 0} C_DIS
LIN {X 403.092, Y 488.654, Z 271.276, A 0, B 90, C -86.012, E1 0, E2 0, E3 0, E4 0} C_DIS
LIN {X 401.874, Y 488.241, Z 270.579, A 0, B 90, C -86.084, E1 0, E2 0, E3 0, E4 0} C_DIS
LIN {X 400.658, Y 487.82, Z 269.883, A 0, B 90, C -86.156, E1 0, E2 0, E3 0, E4 0} C_DIS
LIN {X 399.443, Y 487.392, Z 269.188, A 0, B 90, C -86.228, E1 0, E2 0, E3 0, E4 0} C_DIS
LIN {X 398.231, Y 486.956, Z 268.495, A 0, B 90, C -86.3, E1 0, E2 0, E3 0, E4 0} C_DIS
LIN {X 397.021, Y 486.512, Z 267.802, A 0, B 90, C -86.372, E1 0, E2 0, E3 0, E4 0} C_DIS
LIN {X 395.813, Y 486.061, Z 267.111, A 0, B 90, C -86.444, E1 0, E2 0, E3 0, E4 0} C_DIS
LIN {X 394.607, Y 485.602, Z 266.421, A 0, B 90, C -86.516, E1 0, E2 0, E3 0, E4 0} C_DIS
LIN {X 393.404, Y 485.135, Z 265.733, A 0, B 90, C -86.587, E1 0, E2 0, E3 0, E4 0} C_DIS
LIN {X 392.202, Y 484.661, Z 265.045, A 0, B 90, C -86.659, E1 0, E2 0, E3 0, E4 0} C_DIS
LIN {X 391.003, Y 484.18, Z 264.359, A 0, B 90, C -86.73, E1 0, E2 0, E3 0, E4 0} C_DIS
LIN {X 389.806, Y 483.691, Z 263.674, A 0, B 90, C -86.802, E1 0, E2 0, E3 0, E4 0} C_DIS
LIN {X 388.612, Y 483.194, Z 262.991, A 0, B 90, C -86.873, E1 0, E2 0, E3 0, E4 0} C_DIS
LIN {X 387.42, Y 482.69, Z 262.309, A 0, B 90, C -86.944, E1 0, E2 0, E3 0, E4 0} C_DIS
LIN {X 386.23, Y 482.179, Z 261.628, A 0, B 90, C -87.015, E1 0, E2 0, E3 0, E4 0} C_DIS
LIN {X 385.043, Y 481.66, Z 260.949, A 0, B 90, C -87.087, E1 0, E2 0, E3 0, E4 0} C_DIS
LIN {X 383.858, Y 481.133, Z 260.271, A 0, B 90, C -87.158, E1 0, E2 0, E3 0, E4 0} C_DIS
LIN {X 382.675, Y 480.599, Z 259.594, A 0, B 90, C -87.228, E1 0, E2 0, E3 0, E4 0} C_DIS
LIN {X 381.496, Y 480.058, Z 258.919, A 0, B 90, C -87.299, E1 0, E2 0, E3 0, E4 0} C_DIS
LIN {X 380.318, Y 479.509, Z 258.246, A 0, B 90, C -87.37, E1 0, E2 0, E3 0, E4 0} C_DIS
LIN {X 379.144, Y 478.953, Z 257.574, A 0, B 90, C -87.441, E1 0, E2 0, E3 0, E4 0} C_DIS
LIN {X 377.972, Y 478.389, Z 256.903, A 0, B 90, C -87.511, E1 0, E2 0, E3 0, E4 0} C_DIS
LIN {X 376.803, Y 477.818, Z 256.234, A 0, B 90, C -87.582, E1 0, E2 0, E3 0, E4 0} C_DIS
LIN {X 375.636, Y 477.24, Z 255.567, A 0, B 90, C -87.652, E1 0, E2 0, E3 0, E4 0} C_DIS
LIN {X 374.473, Y 476.654, Z 254.901, A 0, B 90, C -87.722, E1 0, E2 0, E3 0, E4 0} C_DIS
LIN {X 373.312, Y 476.061, Z 254.236, A 0, B 90, C -87.793, E1 0, E2 0, E3 0, E4 0} C_DIS
LIN {X 372.153, Y 475.461, Z 253.574, A 0, B 90, C -87.863, E1 0, E2 0, E3 0, E4 0} C_DIS
LIN {X 370.998, Y 474.854, Z 252.913, A 0, B 90, C -87.933, E1 0, E2 0, E3 0, E4 0} C_DIS
LIN {X 369.846, Y 474.239, Z 252.253, A 0, B 90, C -88.003, E1 0, E2 0, E3 0, E4 0} C_DIS
LIN {X 368.696, Y 473.617, Z 251.596, A 0, B 90, C -88.072, E1 0, E2 0, E3 0, E4 0} C_DIS
LIN {X 367.55, Y 472.988, Z 250.94, A 0, B 90, C -88.142, E1 0, E2 0, E3 0, E4 0} C_DIS
LIN {X 366.406, Y 472.351, Z 250.285, A 0, B 90, C -88.212, E1 0, E2 0, E3 0, E4 0} C_DIS
LIN {X 365.266, Y 471.708, Z 249.633, A 0, B 90, C -88.281, E1 0, E2 0, E3 0, E4 0} C_DIS
LIN {X 364.129, Y 471.057, Z 248.982, A 0, B 90, C -88.35, E1 0, E2 0, E3 0, E4 0} C_DIS
LIN {X 362.994, Y 470.399, Z 248.333, A 0, B 90, C -88.42, E1 0, E2 0, E3 0, E4 0} C_DIS
LIN {X 361.863, Y 469.734, Z 247.686, A 0, B 90, C -88.489, E1 0, E2 0, E3 0, E4 0} C_DIS
LIN {X 360.735, Y 469.062, Z 247.041, A 0, B 90, C -88.558, E1 0, E2 0, E3 0, E4 0} C_DIS
LIN {X 359.61, Y 468.383, Z 246.397, A 0, B 90, C -88.627, E1 0, E2 0, E3 0, E4 0} C_DIS
LIN {X 358.489, Y 467.697, Z 245.755, A 0, B 90, C -88.696, E1 0, E2 0, E3 0, E4 0} C_DIS
LIN {X 357.371, Y 467.003, Z 245.115, A 0, B 90, C -88.765, E1 0, E2 0, E3 0, E4 0} C_DIS
LIN {X 356.256, Y 466.303, Z 244.477, A 0, B 90, C -88.833, E1 0, E2 0, E3 0, E4 0} C_DIS
LIN {X 355.144, Y 465.596, Z 243.841, A 0, B 90, C -88.902, E1 0, E2 0, E3 0, E4 0} C_DIS
LIN {X 354.036, Y 464.881, Z 243.207, A 0, B 90, C -88.97, E1 0, E2 0, E3 0, E4 0} C_DIS
LIN {X 352.931, Y 464.16, Z 242.575, A 0, B 90, C -89.039, E1 0, E2 0, E3 0, E4 0} C_DIS
LIN {X 351.829, Y 463.432, Z 241.945, A 0, B 90, C -89.107, E1 0, E2 0, E3 0, E4 0} C_DIS
LIN {X 350.732, Y 462.697, Z 241.317, A 0, B 90, C -89.175, E1 0, E2 0, E3 0, E4 0} C_DIS
LIN {X 349.637, Y 461.955, Z 240.69, A 0, B 90, C -89.243, E1 0, E2 0, E3 0, E4 0} C_DIS
LIN {X 348.546, Y 461.206, Z 240.066, A 0, B 90, C -89.311, E1 0, E2 0, E3 0, E4 0} C_DIS
LIN {X 347.459, Y 460.45, Z 239.444, A 0, B 90, C -89.379, E1 0, E2 0, E3 0, E4 0} C_DIS
LIN {X 346.375, Y 459.687, Z 238.824, A 0, B 90, C -89.446, E1 0, E2 0, E3 0, E4 0} C_DIS
LIN {X 345.295, Y 458.918, Z 238.206, A 0, B 90, C -89.514, E1 0, E2 0, E3 0, E4 0} C_DIS
LIN {X 344.218, Y 458.142, Z 237.59, A 0, B 90, C -89.581, E1 0, E2 0, E3 0, E4 0} C_DIS
LIN {X 343.146, Y 457.359, Z 236.976, A 0, B 90, C -89.649, E1 0, E2 0, E3 0, E4 0} C_DIS
LIN {X 342.077, Y 456.569, Z 236.365, A 0, B 90, C -89.716, E1 0, E2 0, E3 0, E4 0} C_DIS
LIN {X 341.011, Y 455.773, Z 235.755, A 0, B 90, C -89.783, E1 0, E2 0, E3 0, E4 0} C_DIS
LIN {X 339.95, Y 454.97, Z 235.148, A 0, B 90, C -89.85, E1 0, E2 0, E3 0, E4 0} C_DIS
LIN {X 338.892, Y 454.16, Z 234.542, A 0, B 90, C -89.917, E1 0, E2 0, E3 0, E4 0} C_DIS
LIN {X 337.838, Y 453.344, Z 233.939, A 0, B 90, C -89.983, E1 0, E2 0, E3 0, E4 0} C_DIS
LIN {X 336.788, Y 452.521, Z 233.339, A 0, B 90, C -90.05, E1 0, E2 0, E3 0, E4 0} C_DIS
LIN {X 335.742, Y 451.691, Z 232.74, A 0, B 90, C -90.116, E1 0, E2 0, E3 0, E4 0} C_DIS
LIN {X 334.7, Y 450.855, Z 232.144, A 0, B 90, C -90.183, E1 0, E2 0, E3 0, E4 0} C_DIS
LIN {X 333.662, Y 450.012, Z 231.55, A 0, B 90, C -90.249, E1 0, E2 0, E3 0, E4 0} C_DIS
LIN {X 332.628, Y 449.163, Z 230.958, A 0, B 90, C -90.315, E1 0, E2 0, E3 0, E4 0} C_DIS
LIN {X 331.598, Y 448.308, Z 230.369, A 0, B 90, C -90.381, E1 0, E2 0, E3 0, E4 0} C_DIS
LIN {X 330.572, Y 447.445, Z 229.782, A 0, B 90, C -90.447, E1 0, E2 0, E3 0, E4 0} C_DIS
LIN {X 329.55, Y 446.577, Z 229.197, A 0, B 90, C -90.512, E1 0, E2 0, E3 0, E4 0} C_DIS
LIN {X 328.532, Y 445.702, Z 228.615, A 0, B 90, C -90.578, E1 0, E2 0, E3 0, E4 0} C_DIS
LIN {X 327.519, Y 444.82, Z 228.035, A 0, B 90, C -90.643, E1 0, E2 0, E3 0, E4 0} C_DIS
LIN {X 326.509, Y 443.933, Z 227.457, A 0, B 90, C -90.708, E1 0, E2 0, E3 0, E4 0} C_DIS
LIN {X 325.504, Y 443.039, Z 226.882, A 0, B 90, C -90.774, E1 0, E2 0, E3 0, E4 0} C_DIS
LIN {X 324.503, Y 442.138, Z 226.309, A 0, B 90, C -90.838, E1 0, E2 0, E3 0, E4 0} C_DIS
LIN {X 323.506, Y 441.232, Z 225.739, A 0, B 90, C -90.903, E1 0, E2 0, E3 0, E4 0} C_DIS
LIN {X 322.514, Y 440.319, Z 225.171, A 0, B 90, C -90.968, E1 0, E2 0, E3 0, E4 0} C_DIS
LIN {X 321.526, Y 439.399, Z 224.606, A 0, B 90, C -91.033, E1 0, E2 0, E3 0, E4 0} C_DIS
LIN {X 320.542, Y 438.474, Z 224.043, A 0, B 90, C -91.097, E1 0, E2 0, E3 0, E4 0} C_DIS
LIN {X 319.563, Y 437.543, Z 223.483, A 0, B 90, C -91.161, E1 0, E2 0, E3 0, E4 0} C_DIS
LIN {X 318.588, Y 436.605, Z 222.925, A 0, B 90, C -91.225, E1 0, E2 0, E3 0, E4 0} C_DIS
LIN {X 317.618, Y 435.661, Z 222.37, A 0, B 90, C -91.289, E1 0, E2 0, E3 0, E4 0} C_DIS
LIN {X 316.652, Y 434.711, Z 221.817, A 0, B 90, C -91.353, E1 0, E2 0, E3 0, E4 0} C_DIS
LIN {X 315.691, Y 433.755, Z 221.267, A 0, B 90, C -91.417, E1 0, E2 0, E3 0, E4 0} C_DIS
LIN {X 314.734, Y 432.793, Z 220.72, A 0, B 90, C -91.48, E1 0, E2 0, E3 0, E4 0} C_DIS
LIN {X 313.782, Y 431.825, Z 220.175, A 0, B 90, C -91.544, E1 0, E2 0, E3 0, E4 0} C_DIS
LIN {X 312.834, Y 430.851, Z 219.633, A 0, B 90, C -91.607, E1 0, E2 0, E3 0, E4 0} C_DIS
LIN {X 311.891, Y 429.871, Z 219.093, A 0, B 90, C -91.67, E1 0, E2 0, E3 0, E4 0} C_DIS
LIN {X 310.953, Y 428.886, Z 218.556, A 0, B 90, C -91.733, E1 0, E2 0, E3 0, E4 0} C_DIS
LIN {X 310.019, Y 427.894, Z 218.022, A 0, B 90, C -91.796, E1 0, E2 0, E3 0, E4 0} C_DIS
LIN {X 309.09, Y 426.896, Z 217.49, A 0, B 90, C -91.858, E1 0, E2 0, E3 0, E4 0} C_DIS
LIN {X 308.166, Y 425.893, Z 216.962, A 0, B 90, C -91.921, E1 0, E2 0, E3 0, E4 0} C_DIS
LIN {X 307.246, Y 424.884, Z 216.436, A 0, B 90, C -91.983, E1 0, E2 0, E3 0, E4 0} C_DIS
LIN {X 306.332, Y 423.869, Z 215.912, A 0, B 90, C -92.045, E1 0, E2 0, E3 0, E4 0} C_DIS
LIN {X 305.422, Y 422.848, Z 215.392, A 0, B 90, C -92.107, E1 0, E2 0, E3 0, E4 0} C_DIS
LIN {X 304.517, Y 421.822, Z 214.874, A 0, B 90, C -92.169, E1 0, E2 0, E3 0, E4 0} C_DIS
LIN {X 303.617, Y 420.79, Z 214.359, A 0, B 90, C -92.231, E1 0, E2 0, E3 0, E4 0} C_DIS
LIN {X 302.721, Y 419.752, Z 213.847, A 0, B 90, C -92.292, E1 0, E2 0, E3 0, E4 0} C_DIS
LIN {X 301.831, Y 418.709, Z 213.337, A 0, B 90, C -92.353, E1 0, E2 0, E3 0, E4 0} C_DIS
LIN {X 300.946, Y 417.66, Z 212.831, A 0, B 90, C -92.414, E1 0, E2 0, E3 0, E4 0} C_DIS
LIN {X 300.066, Y 416.605, Z 212.327, A 0, B 90, C -92.475, E1 0, E2 0, E3 0, E4 0} C_DIS
LIN {X 299.19, Y 415.545, Z 211.826, A 0, B 90, C -92.536, E1 0, E2 0, E3 0, E4 0} C_DIS
LIN {X 298.32, Y 414.48, Z 211.328, A 0, B 90, C -92.597, E1 0, E2 0, E3 0, E4 0} C_DIS
LIN {X 297.455, Y 413.409, Z 210.833, A 0, B 90, C -92.657, E1 0, E2 0, E3 0, E4 0} C_DIS
LIN {X 296.595, Y 412.333, Z 210.341, A 0, B 90, C -92.718, E1 0, E2 0, E3 0, E4 0} C_DIS
LIN {X 295.74, Y 411.251, Z 209.852, A 0, B 90, C -92.778, E1 0, E2 0, E3 0, E4 0} C_DIS
LIN {X 294.89, Y 410.164, Z 209.365, A 0, B 90, C -92.838, E1 0, E2 0, E3 0, E4 0} C_DIS
LIN {X 294.045, Y 409.071, Z 208.882, A 0, B 90, C -92.897, E1 0, E2 0, E3 0, E4 0} C_DIS
LIN {X 293.205, Y 407.973, Z 208.402, A 0, B 90, C -92.957, E1 0, E2 0, E3 0, E4 0} C_DIS
LIN {X 292.371, Y 406.87, Z 207.924, A 0, B 90, C -93.016, E1 0, E2 0, E3 0, E4 0} C_DIS
LIN {X 291.542, Y 405.762, Z 207.45, A 0, B 90, C -93.075, E1 0, E2 0, E3 0, E4 0} C_DIS
LIN {X 290.718, Y 404.649, Z 206.979, A 0, B 90, C -93.134, E1 0, E2 0, E3 0, E4 0} C_DIS
LIN {X 289.9, Y 403.53, Z 206.51, A 0, B 90, C -93.193, E1 0, E2 0, E3 0, E4 0} C_DIS
LIN {X 289.086, Y 402.406, Z 206.045, A 0, B 90, C -93.252, E1 0, E2 0, E3 0, E4 0} C_DIS
LIN {X 288.279, Y 401.278, Z 205.583, A 0, B 90, C -93.31, E1 0, E2 0, E3 0, E4 0} C_DIS
LIN {X 287.476, Y 400.144, Z 205.123, A 0, B 90, C -93.368, E1 0, E2 0, E3 0, E4 0} C_DIS
LIN {X 286.679, Y 399.005, Z 204.667, A 0, B 90, C -93.426, E1 0, E2 0, E3 0, E4 0} C_DIS
LIN {X 285.887, Y 397.861, Z 204.214, A 0, B 90, C -93.484, E1 0, E2 0, E3 0, E4 0} C_DIS
LIN {X 285.101, Y 396.712, Z 203.764, A 0, B 90, C -93.542, E1 0, E2 0, E3 0, E4 0} C_DIS
LIN {X 284.32, Y 395.558, Z 203.318, A 0, B 90, C -93.599, E1 0, E2 0, E3 0, E4 0} C_DIS
LIN {X 283.545, Y 394.4, Z 202.874, A 0, B 90, C -93.657, E1 0, E2 0, E3 0, E4 0} C_DIS
LIN {X 282.775, Y 393.236, Z 202.434, A 0, B 90, C -93.714, E1 0, E2 0, E3 0, E4 0} C_DIS
LIN {X 282.01, Y 392.068, Z 201.996, A 0, B 90, C -93.771, E1 0, E2 0, E3 0, E4 0} C_DIS
LIN {X 281.252, Y 390.894, Z 201.562, A 0, B 90, C -93.827, E1 0, E2 0, E3 0, E4 0} C_DIS
LIN {X 280.498, Y 389.716, Z 201.131, A 0, B 90, C -93.884, E1 0, E2 0, E3 0, E4 0} C_DIS
LIN {X 279.751, Y 388.534, Z 200.703, A 0, B 90, C -93.94, E1 0, E2 0, E3 0, E4 0} C_DIS
LIN {X 279.009, Y 387.346, Z 200.279, A 0, B 90, C -93.996, E1 0, E2 0, E3 0, E4 0} C_DIS
LIN {X 278.272, Y 386.155, Z 199.857, A 0, B 90, C -94.052, E1 0, E2 0, E3 0, E4 0} C_DIS
LIN {X 277.542, Y 384.958, Z 199.439, A 0, B 90, C -94.107, E1 0, E2 0, E3 0, E4 0} C_DIS
LIN {X 276.817, Y 383.757, Z 199.024, A 0, B 90, C -94.163, E1 0, E2 0, E3 0, E4 0} C_DIS
LIN {X 276.097, Y 382.551, Z 198.613, A 0, B 90, C -94.218, E1 0, E2 0, E3 0, E4 0} C_DIS
LIN {X 275.384, Y 381.341, Z 198.205, A 0, B 90, C -94.273, E1 0, E2 0, E3 0, E4 0} C_DIS
LIN {X 274.676, Y 380.126, Z 197.8, A 0, B 90, C -94.328, E1 0, E2 0, E3 0, E4 0} C_DIS
LIN {X 273.974, Y 378.907, Z 197.398, A 0, B 90, C -94.382, E1 0, E2 0, E3 0, E4 0} C_DIS
LIN {X 273.277, Y 377.683, Z 196.999, A 0, B 90, C -94.436, E1 0, E2 0, E3 0, E4 0} C_DIS
LIN {X 272.587, Y 376.456, Z 196.604, A 0, B 90, C -94.491, E1 0, E2 0, E3 0, E4 0} C_DIS
LIN {X 271.902, Y 375.223, Z 196.213, A 0, B 90, C -94.544, E1 0, E2 0, E3 0, E4 0} C_DIS
LIN {X 271.223, Y 373.987, Z 195.824, A 0, B 90, C -94.598, E1 0, E2 0, E3 0, E4 0} C_DIS
LIN {X 270.55, Y 372.746, Z 195.439, A 0, B 90, C -94.651, E1 0, E2 0, E3 0, E4 0} C_DIS
LIN {X 269.883, Y 371.501, Z 195.057, A 0, B 90, C -94.705, E1 0, E2 0, E3 0, E4 0} C_DIS
LIN {X 269.222, Y 370.252, Z 194.679, A 0, B 90, C -94.758, E1 0, E2 0, E3 0, E4 0} C_DIS
LIN {X 268.567, Y 368.999, Z 194.304, A 0, B 90, C -94.81, E1 0, E2 0, E3 0, E4 0} C_DIS
LIN {X 267.918, Y 367.741, Z 193.933, A 0, B 90, C -94.863, E1 0, E2 0, E3 0, E4 0} C_DIS
LIN {X 267.274, Y 366.48, Z 193.565, A 0, B 90, C -94.915, E1 0, E2 0, E3 0, E4 0} C_DIS
LIN {X 266.637, Y 365.214, Z 193.2, A 0, B 90, C -94.967, E1 0, E2 0, E3 0, E4 0} C_DIS
LIN {X 266.006, Y 363.945, Z 192.839, A 0, B 90, C -95.019, E1 0, E2 0, E3 0, E4 0} C_DIS
LIN {X 265.38, Y 362.672, Z 192.481, A 0, B 90, C -95.07, E1 0, E2 0, E3 0, E4 0} C_DIS
LIN {X 264.761, Y 361.394, Z 192.127, A 0, B 90, C -95.121, E1 0, E2 0, E3 0, E4 0} C_DIS
LIN {X 264.148, Y 360.113, Z 191.776, A 0, B 90, C -95.172, E1 0, E2 0, E3 0, E4 0} C_DIS
LIN {X 263.541, Y 358.828, Z 191.428, A 0, B 90, C -95.223, E1 0, E2 0, E3 0, E4 0} C_DIS
LIN {X 262.94, Y 357.539, Z 191.084, A 0, B 90, C -95.274, E1 0, E2 0, E3 0, E4 0} C_DIS
LIN {X 262.345, Y 356.246, Z 190.744, A 0, B 90, C -95.324, E1 0, E2 0, E3 0, E4 0} C_DIS
LIN {X 261.756, Y 354.95, Z 190.407, A 0, B 90, C -95.374, E1 0, E2 0, E3 0, E4 0} C_DIS
LIN {X 261.173, Y 353.65, Z 190.074, A 0, B 90, C -95.424, E1 0, E2 0, E3 0, E4 0} C_DIS
LIN {X 260.597, Y 352.346, Z 189.744, A 0, B 90, C -95.473, E1 0, E2 0, E3 0, E4 0} C_DIS
LIN {X 260.027, Y 351.039, Z 189.418, A 0, B 90, C -95.522, E1 0, E2 0, E3 0, E4 0} C_DIS
LIN {X 259.463, Y 349.728, Z 189.095, A 0, B 90, C -95.571, E1 0, E2 0, E3 0, E4 0} C_DIS
LIN {X 258.905, Y 348.414, Z 188.776, A 0, B 90, C -95.62, E1 0, E2 0, E3 0, E4 0} C_DIS
LIN {X 258.353, Y 347.096, Z 188.46, A 0, B 90, C -95.669, E1 0, E2 0, E3 0, E4 0} C_DIS
LIN {X 257.808, Y 345.775, Z 188.148, A 0, B 90, C -95.717, E1 0, E2 0, E3 0, E4 0} C_DIS
LIN {X 257.269, Y 344.45, Z 187.84, A 0, B 90, C -95.765, E1 0, E2 0, E3 0, E4 0} C_DIS
LIN {X 256.736, Y 343.122, Z 187.535, A 0, B 90, C -95.812, E1 0, E2 0, E3 0, E4 0} C_DIS
LIN {X 256.209, Y 341.791, Z 187.234, A 0, B 90, C -95.86, E1 0, E2 0, E3 0, E4 0} C_DIS
LIN {X 255.689, Y 340.456, Z 186.936, A 0, B 90, C -95.907, E1 0, E2 0, E3 0, E4 0} C_DIS
LIN {X 255.175, Y 339.118, Z 186.642, A 0, B 90, C -95.953, E1 0, E2 0, E3 0, E4 0} C_DIS
LIN {X 254.668, Y 337.777, Z 186.351, A 0, B 90, C -96, E1 0, E2 0, E3 0, E4 0} C_DIS
LIN {X 254.167, Y 336.433, Z 186.065, A 0, B 90, C -96.046, E1 0, E2 0, E3 0, E4 0} C_DIS
LIN {X 253.672, Y 335.085, Z 185.782, A 0, B 90, C -96.092, E1 0, E2 0, E3 0, E4 0} C_DIS
LIN {X 253.184, Y 333.735, Z 185.502, A 0, B 90, C -96.138, E1 0, E2 0, E3 0, E4 0} C_DIS
LIN {X 252.702, Y 332.381, Z 185.226, A 0, B 90, C -96.183, E1 0, E2 0, E3 0, E4 0} C_DIS
LIN {X 252.226, Y 331.024, Z 184.954, A 0, B 90, C -96.228, E1 0, E2 0, E3 0, E4 0} C_DIS
LIN {X 251.757, Y 329.665, Z 184.686, A 0, B 90, C -96.273, E1 0, E2 0, E3 0, E4 0} C_DIS
LIN {X 251.294, Y 328.302, Z 184.421, A 0, B 90, C -96.317, E1 0, E2 0, E3 0, E4 0} C_DIS
LIN {X 250.838, Y 326.937, Z 184.16, A 0, B 90, C -96.362, E1 0, E2 0, E3 0, E4 0} C_DIS
LIN {X 250.388, Y 325.569, Z 183.903, A 0, B 90, C -96.406, E1 0, E2 0, E3 0, E4 0} C_DIS
LIN {X 249.945, Y 324.198, Z 183.649, A 0, B 90, C -96.449, E1 0, E2 0, E3 0, E4 0} C_DIS
LIN {X 249.508, Y 322.824, Z 183.399, A 0, B 90, C -96.492, E1 0, E2 0, E3 0, E4 0} C_DIS
LIN {X 249.078, Y 321.447, Z 183.153, A 0, B 90, C -96.535, E1 0, E2 0, E3 0, E4 0} C_DIS
LIN {X 248.654, Y 320.068, Z 182.911, A 0, B 90, C -96.578, E1 0, E2 0, E3 0, E4 0} C_DIS
LIN {X 248.237, Y 318.686, Z 182.672, A 0, B 90, C -96.62, E1 0, E2 0, E3 0, E4 0} C_DIS
LIN {X 247.827, Y 317.301, Z 182.437, A 0, B 90, C -96.662, E1 0, E2 0, E3 0, E4 0} C_DIS
LIN {X 247.423, Y 315.914, Z 182.206, A 0, B 90, C -96.704, E1 0, E2 0, E3 0, E4 0} C_DIS
LIN {X 247.025, Y 314.525, Z 181.978, A 0, B 90, C -96.746, E1 0, E2 0, E3 0, E4 0} C_DIS
LIN {X 246.634, Y 313.133, Z 181.755, A 0, B 90, C -96.787, E1 0, E2 0, E3 0, E4 0} C_DIS
LIN {X 246.25, Y 311.738, Z 181.535, A 0, B 90, C -96.827, E1 0, E2 0, E3 0, E4 0} C_DIS
LIN {X 245.872, Y 310.341, Z 181.319, A 0, B 90, C -96.868, E1 0, E2 0, E3 0, E4 0} C_DIS
LIN {X 245.501, Y 308.942, Z 181.107, A 0, B 90, C -96.908, E1 0, E2 0, E3 0, E4 0} C_DIS
LIN {X 245.137, Y 307.541, Z 180.898, A 0, B 90, C -96.948, E1 0, E2 0, E3 0, E4 0} C_DIS
LIN {X 244.779, Y 306.137, Z 180.693, A 0, B 90, C -96.987, E1 0, E2 0, E3 0, E4 0} C_DIS
LIN {X 244.428, Y 304.731, Z 180.493, A 0, B 90, C -97.026, E1 0, E2 0, E3 0, E4 0} C_DIS
LIN {X 244.084, Y 303.323, Z 180.295, A 0, B 90, C -97.065, E1 0, E2 0, E3 0, E4 0} C_DIS
LIN {X 243.746, Y 301.912, Z 180.102, A 0, B 90, C -97.103, E1 0, E2 0, E3 0, E4 0} C_DIS
LIN {X 243.415, Y 300.5, Z 179.913, A 0, B 90, C -97.141, E1 0, E2 0, E3 0, E4 0} C_DIS
LIN {X 243.091, Y 299.085, Z 179.727, A 0, B 90, C -97.179, E1 0, E2 0, E3 0, E4 0} C_DIS
LIN {X 242.773, Y 297.669, Z 179.545, A 0, B 90, C -97.216, E1 0, E2 0, E3 0, E4 0} C_DIS
LIN {X 242.462, Y 296.25, Z 179.368, A 0, B 90, C -97.253, E1 0, E2 0, E3 0, E4 0} C_DIS
LIN {X 242.158, Y 294.829, Z 179.193, A 0, B 90, C -97.29, E1 0, E2 0, E3 0, E4 0} C_DIS
LIN {X 241.86, Y 293.407, Z 179.023, A 0, B 90, C -97.326, E1 0, E2 0, E3 0, E4 0} C_DIS
LIN {X 241.57, Y 291.983, Z 178.857, A 0, B 90, C -97.362, E1 0, E2 0, E3 0, E4 0} C_DIS
LIN {X 241.286, Y 290.557, Z 178.694, A 0, B 90, C -97.398, E1 0, E2 0, E3 0, E4 0} C_DIS
LIN {X 241.008, Y 289.129, Z 178.536, A 0, B 90, C -97.433, E1 0, E2 0, E3 0, E4 0} C_DIS
LIN {X 240.738, Y 287.7, Z 178.381, A 0, B 90, C -97.468, E1 0, E2 0, E3 0, E4 0} C_DIS
LIN {X 240.474, Y 286.268, Z 178.23, A 0, B 90, C -97.502, E1 0, E2 0, E3 0, E4 0} C_DIS
LIN {X 240.217, Y 284.836, Z 178.083, A 0, B 90, C -97.537, E1 0, E2 0, E3 0, E4 0} C_DIS
LIN {X 239.967, Y 283.401, Z 177.94, A 0, B 90, C -97.57, E1 0, E2 0, E3 0, E4 0} C_DIS
LIN {X 239.724, Y 281.965, Z 177.801, A 0, B 90, C -97.604, E1 0, E2 0, E3 0, E4 0} C_DIS
LIN {X 239.487, Y 280.528, Z 177.666, A 0, B 90, C -97.637, E1 0, E2 0, E3 0, E4 0} C_DIS
LIN {X 239.258, Y 279.089, Z 177.534, A 0, B 90, C -97.669, E1 0, E2 0, E3 0, E4 0} C_DIS
LIN {X 239.035, Y 277.648, Z 177.407, A 0, B 90, C -97.701, E1 0, E2 0, E3 0, E4 0} C_DIS
LIN {X 238.819, Y 276.207, Z 177.283, A 0, B 90, C -97.733, E1 0, E2 0, E3 0, E4 0} C_DIS
LIN {X 238.61, Y 274.763, Z 177.163, A 0, B 90, C -97.765, E1 0, E2 0, E3 0, E4 0} C_DIS
LIN {X 238.407, Y 273.319, Z 177.048, A 0, B 90, C -97.796, E1 0, E2 0, E3 0, E4 0} C_DIS
LIN {X 238.212, Y 271.873, Z 176.936, A 0, B 90, C -97.826, E1 0, E2 0, E3 0, E4 0} C_DIS
LIN {X 238.023, Y 270.427, Z 176.828, A 0, B 90, C -97.856, E1 0, E2 0, E3 0, E4 0} C_DIS
LIN {X 237.841, Y 268.979, Z 176.724, A 0, B 90, C -97.886, E1 0, E2 0, E3 0, E4 0} C_DIS
LIN {X 237.666, Y 267.529, Z 176.624, A 0, B 90, C -97.916, E1 0, E2 0, E3 0, E4 0} C_DIS
LIN {X 237.498, Y 266.079, Z 176.528, A 0, B 90, C -97.945, E1 0, E2 0, E3 0, E4 0} C_DIS
LIN {X 237.337, Y 264.628, Z 176.435, A 0, B 90, C -97.973, E1 0, E2 0, E3 0, E4 0} C_DIS
LIN {X 237.183, Y 263.176, Z 176.347, A 0, B 90, C -98.001, E1 0, E2 0, E3 0, E4 0} C_DIS
LIN {X 237.036, Y 261.723, Z 176.263, A 0, B 90, C -98.029, E1 0, E2 0, E3 0, E4 0} C_DIS
LIN {X 236.895, Y 260.268, Z 176.182, A 0, B 90, C -98.056, E1 0, E2 0, E3 0, E4 0} C_DIS
LIN {X 236.761, Y 258.813, Z 176.106, A 0, B 90, C -98.083, E1 0, E2 0, E3 0, E4 0} C_DIS
LIN {X 236.635, Y 257.358, Z 176.033, A 0, B 90, C -98.11, E1 0, E2 0, E3 0, E4 0} C_DIS
LIN {X 236.515, Y 255.901, Z 175.965, A 0, B 90, C -98.136, E1 0, E2 0, E3 0, E4 0} C_DIS
LIN {X 236.402, Y 254.444, Z 175.9, A 0, B 90, C -98.161, E1 0, E2 0, E3 0, E4 0} C_DIS
LIN {X 236.296, Y 252.986, Z 175.839, A 0, B 90, C -98.186, E1 0, E2 0, E3 0, E4 0} C_DIS
LIN {X 236.197, Y 251.527, Z 175.783, A 0, B 90, C -98.211, E1 0, E2 0, E3 0, E4 0} C_DIS
LIN {X 236.104, Y 250.068, Z 175.73, A 0, B 90, C -98.235, E1 0, E2 0, E3 0, E4 0} C_DIS
LIN {X 236.019, Y 248.608, Z 175.681, A 0, B 90, C -98.259, E1 0, E2 0, E3 0, E4 0} C_DIS
LIN {X 235.941, Y 247.148, Z 175.636, A 0, B 90, C -98.282, E1 0, E2 0, E3 0, E4 0} C_DIS
LIN {X 235.869, Y 245.687, Z 175.595, A 0, B 90, C -98.305, E1 0, E2 0, E3 0, E4 0} C_DIS
LIN {X 235.805, Y 244.226, Z 175.558, A 0, B 90, C -98.328, E1 0, E2 0, E3 0, E4 0} C_DIS
LIN {X 235.747, Y 242.764, Z 175.525, A 0, B 90, C -98.35, E1 0, E2 0, E3 0, E4 0} C_DIS
LIN {X 235.696, Y 241.303, Z 175.497, A 0, B 90, C -98.371, E1 0, E2 0, E3 0, E4 0} C_DIS
LIN {X 235.653, Y 239.84, Z 175.471, A 0, B 90, C -98.392, E1 0, E2 0, E3 0, E4 0} C_DIS
LIN {X 235.616, Y 238.378, Z 175.45, A 0, B 90, C -98.413, E1 0, E2 0, E3 0, E4 0} C_DIS
LIN {X 235.586, Y 236.915, Z 175.433, A 0, B 90, C -98.433, E1 0, E2 0, E3 0, E4 0} C_DIS
LIN {X 235.563, Y 235.452, Z 175.42, A 0, B 90, C -98.452, E1 0, E2 0, E3 0, E4 0} C_DIS
LIN {X 235.547, Y 233.989, Z 175.411, A 0, B 90, C -98.471, E1 0, E2 0, E3 0, E4 0} C_DIS
LIN {X 235.538, Y 232.526, Z 175.406, A 0, B 90, C -98.49, E1 0, E2 0, E3 0, E4 0} C_DIS
LIN {X 235.536, Y 231.063, Z 175.404, A 0, B 90, C -98.508, E1 0, E2 0, E3 0, E4 0} C_DIS
LIN {X 235.54, Y 229.6, Z 175.407, A 0, B 90, C -98.526, E1 0, E2 0, E3 0, E4 0} C_DIS
LIN {X 235.552, Y 228.137, Z 175.414, A 0, B 90, C -98.543, E1 0, E2 0, E3 0, E4 0} C_DIS
LIN {X 235.571, Y 226.674, Z 175.425, A 0, B 90, C -98.559, E1 0, E2 0, E3 0, E4 0} C_DIS
LIN {X 235.596, Y 225.211, Z 175.439, A 0, B 90, C -98.576, E1 0, E2 0, E3 0, E4 0} C_DIS
LIN {X 235.629, Y 223.749, Z 175.458, A 0, B 90, C -98.591, E1 0, E2 0, E3 0, E4 0} C_DIS
LIN {X 235.668, Y 222.286, Z 175.48, A 0, B 90, C -98.606, E1 0, E2 0, E3 0, E4 0} C_DIS
LIN {X 235.714, Y 220.824, Z 175.507, A 0, B 90, C -98.621, E1 0, E2 0, E3 0, E4 0} C_DIS
LIN {X 235.768, Y 219.363, Z 175.537, A 0, B 90, C -98.635, E1 0, E2 0, E3 0, E4 0} C_DIS
LIN {X 235.828, Y 217.901, Z 175.572, A 0, B 90, C -98.648, E1 0, E2 0, E3 0, E4 0} C_DIS
LIN {X 235.895, Y 216.44, Z 175.61, A 0, B 90, C -98.661, E1 0, E2 0, E3 0, E4 0} C_DIS
LIN {X 235.969, Y 214.98, Z 175.652, A 0, B 90, C -98.674, E1 0, E2 0, E3 0, E4 0} C_DIS
LIN {X 236.05, Y 213.519, Z 175.699, A 0, B 90, C -98.686, E1 0, E2 0, E3 0, E4 0} C_DIS
LIN {X 236.138, Y 212.06, Z 175.749, A 0, B 90, C -98.697, E1 0, E2 0, E3 0, E4 0} C_DIS
LIN {X 236.233, Y 210.601, Z 175.803, A 0, B 90, C -98.708, E1 0, E2 0, E3 0, E4 0} C_DIS
LIN {X 236.334, Y 209.142, Z 175.862, A 0, B 90, C -98.719, E1 0, E2 0, E3 0, E4 0} C_DIS
LIN {X 236.443, Y 207.685, Z 175.924, A 0, B 90, C -98.728, E1 0, E2 0, E3 0, E4 0} C_DIS
LIN {X 236.559, Y 206.228, Z 175.99, A 0, B 90, C -98.737, E1 0, E2 0, E3 0, E4 0} C_DIS
LIN {X 236.681, Y 204.771, Z 176.06, A 0, B 90, C -98.746, E1 0, E2 0, E3 0, E4 0} C_DIS
LIN {X 236.81, Y 203.316, Z 176.134, A 0, B 90, C -98.754, E1 0, E2 0, E3 0, E4 0} C_DIS
LIN {X 236.946, Y 201.861, Z 176.212, A 0, B 90, C -98.762, E1 0, E2 0, E3 0, E4 0} C_DIS
LIN {X 237.09, Y 200.408, Z 176.294, A 0, B 90, C -98.769, E1 0, E2 0, E3 0, E4 0} C_DIS
LIN {X 237.239, Y 198.955, Z 176.379, A 0, B 90, C -98.775, E1 0, E2 0, E3 0, E4 0} C_DIS
LIN {X 237.396, Y 197.503, Z 176.469, A 0, B 90, C -98.781, E1 0, E2 0, E3 0, E4 0} C_DIS
LIN {X 237.56, Y 196.052, Z 176.563, A 0, B 90, C -98.786, E1 0, E2 0, E3 0, E4 0} C_DIS
LIN {X 237.731, Y 194.602, Z 176.66, A 0, B 90, C -98.791, E1 0, E2 0, E3 0, E4 0} C_DIS
LIN {X 237.908, Y 193.153, Z 176.762, A 0, B 90, C -98.795, E1 0, E2 0, E3 0, E4 0} C_DIS
LIN {X 238.093, Y 191.706, Z 176.867, A 0, B 90, C -98.798, E1 0, E2 0, E3 0, E4 0} C_DIS
LIN {X 238.284, Y 190.259, Z 176.977, A 0, B 90, C -98.801, E1 0, E2 0, E3 0, E4 0} C_DIS
LIN {X 238.482, Y 188.814, Z 177.09, A 0, B 90, C -98.803, E1 0, E2 0, E3 0, E4 0} C_DIS
LIN {X 238.687, Y 187.37, Z 177.207, A 0, B 90, C -98.805, E1 0, E2 0, E3 0, E4 0} C_DIS
LIN {X 238.898, Y 185.928, Z 177.329, A 0, B 90, C -98.806, E1 0, E2 0, E3 0, E4 0} C_DIS
LIN {X 239.117, Y 184.487, Z 177.454, A 0, B 90, C -98.806, E1 0, E2 0, E3 0, E4 0} C_DIS
LIN {X 239.342, Y 183.047, Z 177.583, A 0, B 90, C -98.806, E1 0, E2 0, E3 0, E4 0} C_DIS
LIN {X 239.575, Y 181.608, Z 177.715, A 0, B 90, C -98.805, E1 0, E2 0, E3 0, E4 0} C_DIS
LIN {X 239.814, Y 180.171, Z 177.852, A 0, B 90, C -98.804, E1 0, E2 0, E3 0, E4 0} C_DIS
LIN {X 240.059, Y 178.736, Z 177.993, A 0, B 90, C -98.802, E1 0, E2 0, E3 0, E4 0} C_DIS
LIN {X 240.312, Y 177.302, Z 178.137, A 0, B 90, C -98.799, E1 0, E2 0, E3 0, E4 0} C_DIS
LIN {X 240.571, Y 175.87, Z 178.286, A 0, B 90, C -98.796, E1 0, E2 0, E3 0, E4 0} C_DIS
LIN {X 240.838, Y 174.439, Z 178.438, A 0, B 90, C -98.792, E1 0, E2 0, E3 0, E4 0} C_DIS
LIN {X 241.111, Y 173.01, Z 178.594, A 0, B 90, C -98.787, E1 0, E2 0, E3 0, E4 0} C_DIS
LIN {X 241.39, Y 171.583, Z 178.754, A 0, B 90, C -98.782, E1 0, E2 0, E3 0, E4 0} C_DIS
LIN {X 241.677, Y 170.158, Z 178.918, A 0, B 90, C -98.776, E1 0, E2 0, E3 0, E4 0} C_DIS
LIN {X 241.97, Y 168.734, Z 179.086, A 0, B 90, C -98.769, E1 0, E2 0, E3 0, E4 0} C_DIS
LIN {X 242.27, Y 167.313, Z 179.258, A 0, B 90, C -98.762, E1 0, E2 0, E3 0, E4 0} C_DIS
LIN {X 242.577, Y 165.893, Z 179.433, A 0, B 90, C -98.754, E1 0, E2 0, E3 0, E4 0} C_DIS
LIN {X 242.89, Y 164.475, Z 179.613, A 0, B 90, C -98.745, E1 0, E2 0, E3 0, E4 0} C_DIS
LIN {X 243.21, Y 163.059, Z 179.796, A 0, B 90, C -98.736, E1 0, E2 0, E3 0, E4 0} C_DIS
LIN {X 243.537, Y 161.645, Z 179.983, A 0, B 90, C -98.726, E1 0, E2 0, E3 0, E4 0} C_DIS
LIN {X 243.871, Y 160.234, Z 180.174, A 0, B 90, C -98.715, E1 0, E2 0, E3 0, E4 0} C_DIS
LIN {X 244.211, Y 158.824, Z 180.368, A 0, B 90, C -98.704, E1 0, E2 0, E3 0, E4 0} C_DIS
LIN {X 244.558, Y 157.417, Z 180.567, A 0, B 90, C -98.692, E1 0, E2 0, E3 0, E4 0} C_DIS
LIN {X 244.911, Y 156.012, Z 180.769, A 0, B 90, C -98.679, E1 0, E2 0, E3 0, E4 0} C_DIS
LIN {X 245.272, Y 154.609, Z 180.975, A 0, B 90, C -98.665, E1 0, E2 0, E3 0, E4 0} C_DIS
LIN {X 245.638, Y 153.208, Z 181.185, A 0, B 90, C -98.651, E1 0, E2 0, E3 0, E4 0} C_DIS
LIN {X 246.012, Y 151.809, Z 181.399, A 0, B 90, C -98.636, E1 0, E2 0, E3 0, E4 0} C_DIS
LIN {X 246.392, Y 150.413, Z 181.616, A 0, B 90, C -98.621, E1 0, E2 0, E3 0, E4 0} C_DIS
LIN {X 246.779, Y 149.02, Z 181.838, A 0, B 90, C -98.604, E1 0, E2 0, E3 0, E4 0} C_DIS
LIN {X 247.172, Y 147.629, Z 182.063, A 0, B 90, C -98.587, E1 0, E2 0, E3 0, E4 0} C_DIS
LIN {X 247.572, Y 146.24, Z 182.291, A 0, B 90, C -98.569, E1 0, E2 0, E3 0, E4 0} C_DIS
LIN {X 247.978, Y 144.854, Z 182.524, A 0, B 90, C -98.551, E1 0, E2 0, E3 0, E4 0} C_DIS
LIN {X 248.392, Y 143.47, Z 182.76, A 0, B 90, C -98.531, E1 0, E2 0, E3 0, E4 0} C_DIS
LIN {X 248.811, Y 142.09, Z 183, A 0, B 90, C -98.511, E1 0, E2 0, E3 0, E4 0} C_DIS
LIN {X 249.237, Y 140.711, Z 183.244, A 0, B 90, C -98.491, E1 0, E2 0, E3 0, E4 0} C_DIS
LIN {X 249.67, Y 139.336, Z 183.492, A 0, B 90, C -98.469, E1 0, E2 0, E3 0, E4 0} C_DIS
LIN {X 250.109, Y 137.963, Z 183.743, A 0, B 90, C -98.447, E1 0, E2 0, E3 0, E4 0} C_DIS
LIN {X 250.555, Y 136.593, Z 183.998, A 0, B 90, C -98.423, E1 0, E2 0, E3 0, E4 0} C_DIS
LIN {X 251.007, Y 135.226, Z 184.257, A 0, B 90, C -98.4, E1 0, E2 0, E3 0, E4 0} C_DIS
LIN {X 251.465, Y 133.861, Z 184.519, A 0, B 90, C -98.375, E1 0, E2 0, E3 0, E4 0} C_DIS
LIN {X 251.931, Y 132.5, Z 184.785, A 0, B 90, C -98.35, E1 0, E2 0, E3 0, E4 0} C_DIS
LIN {X 252.402, Y 131.141, Z 185.055, A 0, B 90, C -98.323, E1 0, E2 0, E3 0, E4 0} C_DIS
LIN {X 252.88, Y 129.786, Z 185.328, A 0, B 90, C -98.296, E1 0, E2 0, E3 0, E4 0} C_DIS
LIN {X 253.364, Y 128.433, Z 185.606, A 0, B 90, C -98.268, E1 0, E2 0, E3 0, E4 0} C_DIS
LIN {X 253.855, Y 127.084, Z 185.886, A 0, B 90, C -98.24, E1 0, E2 0, E3 0, E4 0} C_DIS
LIN {X 254.352, Y 125.738, Z 186.171, A 0, B 90, C -98.21, E1 0, E2 0, E3 0, E4 0} C_DIS
LIN {X 254.856, Y 124.395, Z 186.459, A 0, B 90, C -98.18, E1 0, E2 0, E3 0, E4 0} C_DIS
LIN {X 255.366, Y 123.055, Z 186.751, A 0, B 90, C -98.149, E1 0, E2 0, E3 0, E4 0} C_DIS
LIN {X 255.882, Y 121.718, Z 187.046, A 0, B 90, C -98.117, E1 0, E2 0, E3 0, E4 0} C_DIS
LIN {X 256.404, Y 120.384, Z 187.345, A 0, B 90, C -98.085, E1 0, E2 0, E3 0, E4 0} C_DIS
LIN {X 256.933, Y 119.054, Z 187.648, A 0, B 90, C -98.051, E1 0, E2 0, E3 0, E4 0} C_DIS
LIN {X 257.468, Y 117.727, Z 187.954, A 0, B 90, C -98.017, E1 0, E2 0, E3 0, E4 0} C_DIS
LIN {X 258.01, Y 116.404, Z 188.264, A 0, B 90, C -97.982, E1 0, E2 0, E3 0, E4 0} C_DIS
LIN {X 258.557, Y 115.084, Z 188.577, A 0, B 90, C -97.946, E1 0, E2 0, E3 0, E4 0} C_DIS
LIN {X 259.111, Y 113.767, Z 188.894, A 0, B 90, C -97.909, E1 0, E2 0, E3 0, E4 0} C_DIS
LIN {X 259.672, Y 112.454, Z 189.214, A 0, B 90, C -97.871, E1 0, E2 0, E3 0, E4 0} C_DIS
LIN {X 260.238, Y 111.145, Z 189.539, A 0, B 90, C -97.833, E1 0, E2 0, E3 0, E4 0} C_DIS
LIN {X 260.811, Y 109.839, Z 189.866, A 0, B 90, C -97.793, E1 0, E2 0, E3 0, E4 0} C_DIS
LIN {X 261.389, Y 108.537, Z 190.197, A 0, B 90, C -97.753, E1 0, E2 0, E3 0, E4 0} C_DIS
LIN {X 261.974, Y 107.238, Z 190.532, A 0, B 90, C -97.712, E1 0, E2 0, E3 0, E4 0} C_DIS
LIN {X 262.565, Y 105.943, Z 190.87, A 0, B 90, C -97.67, E1 0, E2 0, E3 0, E4 0} C_DIS
LIN {X 263.162, Y 104.652, Z 191.212, A 0, B 90, C -97.627, E1 0, E2 0, E3 0, E4 0} C_DIS
LIN {X 263.766, Y 103.364, Z 191.557, A 0, B 90, C -97.583, E1 0, E2 0, E3 0, E4 0} C_DIS
LIN {X 264.375, Y 102.081, Z 191.906, A 0, B 90, C -97.539, E1 0, E2 0, E3 0, E4 0} C_DIS
LIN {X 264.991, Y 100.801, Z 192.258, A 0, B 90, C -97.493, E1 0, E2 0, E3 0, E4 0} C_DIS
LIN {X 265.612, Y 99.525, Z 192.613, A 0, B 90, C -97.447, E1 0, E2 0, E3 0, E4 0} C_DIS
LIN {X 266.24, Y 98.253, Z 192.973, A 0, B 90, C -97.399, E1 0, E2 0, E3 0, E4 0} C_DIS
LIN {X 266.873, Y 96.985, Z 193.335, A 0, B 90, C -97.351, E1 0, E2 0, E3 0, E4 0} C_DIS
LIN {X 267.513, Y 95.721, Z 193.701, A 0, B 90, C -97.302, E1 0, E2 0, E3 0, E4 0} C_DIS
LIN {X 268.158, Y 94.461, Z 194.07, A 0, B 90, C -97.252, E1 0, E2 0, E3 0, E4 0} C_DIS
LIN {X 268.81, Y 93.205, Z 194.443, A 0, B 90, C -97.201, E1 0, E2 0, E3 0, E4 0} C_DIS
LIN {X 269.467, Y 91.954, Z 194.819, A 0, B 90, C -97.149, E1 0, E2 0, E3 0, E4 0} C_DIS
LIN {X 270.131, Y 90.706, Z 195.199, A 0, B 90, C -97.096, E1 0, E2 0, E3 0, E4 0} C_DIS
LIN {X 270.8, Y 89.463, Z 195.582, A 0, B 90, C -97.043, E1 0, E2 0, E3 0, E4 0} C_DIS
LIN {X 271.475, Y 88.223, Z 195.968, A 0, B 90, C -96.988, E1 0, E2 0, E3 0, E4 0} C_DIS
LIN {X 272.156, Y 86.989, Z 196.358, A 0, B 90, C -96.933, E1 0, E2 0, E3 0, E4 0} C_DIS
LIN {X 272.843, Y 85.758, Z 196.751, A 0, B 90, C -96.876, E1 0, E2 0, E3 0, E4 0} C_DIS
LIN {X 273.536, Y 84.532, Z 197.147, A 0, B 90, C -96.819, E1 0, E2 0, E3 0, E4 0} C_DIS
LIN {X 274.234, Y 83.31, Z 197.547, A 0, B 90, C -96.76, E1 0, E2 0, E3 0, E4 0} C_DIS
LIN {X 274.938, Y 82.092, Z 197.95, A 0, B 90, C -96.701, E1 0, E2 0, E3 0, E4 0} C_DIS
LIN {X 275.648, Y 80.879, Z 198.356, A 0, B 90, C -96.641, E1 0, E2 0, E3 0, E4 0} C_DIS
LIN {X 276.364, Y 79.671, Z 198.765, A 0, B 90, C -96.579, E1 0, E2 0, E3 0, E4 0} C_DIS
LIN {X 277.085, Y 78.467, Z 199.178, A 0, B 90, C -96.517, E1 0, E2 0, E3 0, E4 0} C_DIS
LIN {X 277.813, Y 77.267, Z 199.594, A 0, B 90, C -96.454, E1 0, E2 0, E3 0, E4 0} C_DIS
LIN {X 278.545, Y 76.072, Z 200.014, A 0, B 90, C -96.39, E1 0, E2 0, E3 0, E4 0} C_DIS
LIN {X 279.284, Y 74.882, Z 200.436, A 0, B 90, C -96.325, E1 0, E2 0, E3 0, E4 0} C_DIS
LIN {X 280.028, Y 73.696, Z 200.862, A 0, B 90, C -96.259, E1 0, E2 0, E3 0, E4 0} C_DIS
LIN {X 280.778, Y 72.516, Z 201.291, A 0, B 90, C -96.191, E1 0, E2 0, E3 0, E4 0} C_DIS
LIN {X 281.533, Y 71.339, Z 201.723, A 0, B 90, C -96.123, E1 0, E2 0, E3 0, E4 0} C_DIS
LIN {X 282.294, Y 70.168, Z 202.158, A 0, B 90, C -96.054, E1 0, E2 0, E3 0, E4 0} C_DIS
LIN {X 283.06, Y 69.001, Z 202.597, A 0, B 90, C -95.984, E1 0, E2 0, E3 0, E4 0} C_DIS
LIN {X 283.832, Y 67.84, Z 203.039, A 0, B 90, C -95.913, E1 0, E2 0, E3 0, E4 0} C_DIS
LIN {X 284.61, Y 66.683, Z 203.483, A 0, B 90, C -95.841, E1 0, E2 0, E3 0, E4 0} C_DIS
LIN {X 285.392, Y 65.531, Z 203.931, A 0, B 90, C -95.768, E1 0, E2 0, E3 0, E4 0} C_DIS
LIN {X 286.181, Y 64.384, Z 204.382, A 0, B 90, C -95.694, E1 0, E2 0, E3 0, E4 0} C_DIS
LIN {X 286.975, Y 63.242, Z 204.837, A 0, B 90, C -95.619, E1 0, E2 0, E3 0, E4 0} C_DIS
LIN {X 287.774, Y 62.105, Z 205.294, A 0, B 90, C -95.543, E1 0, E2 0, E3 0, E4 0} C_DIS
LIN {X 288.578, Y 60.973, Z 205.754, A 0, B 90, C -95.466, E1 0, E2 0, E3 0, E4 0} C_DIS
LIN {X 289.388, Y 59.846, Z 206.217, A 0, B 90, C -95.388, E1 0, E2 0, E3 0, E4 0} C_DIS
LIN {X 290.203, Y 58.724, Z 206.684, A 0, B 90, C -95.309, E1 0, E2 0, E3 0, E4 0} C_DIS
LIN {X 291.024, Y 57.607, Z 207.153, A 0, B 90, C -95.229, E1 0, E2 0, E3 0, E4 0} C_DIS
LIN {X 291.85, Y 56.496, Z 207.626, A 0, B 90, C -95.148, E1 0, E2 0, E3 0, E4 0} C_DIS
LIN {X 292.681, Y 55.389, Z 208.101, A 0, B 90, C -95.066, E1 0, E2 0, E3 0, E4 0} C_DIS
LIN {X 293.517, Y 54.288, Z 208.58, A 0, B 90, C -94.983, E1 0, E2 0, E3 0, E4 0} C_DIS
LIN {X 294.358, Y 53.192, Z 209.061, A 0, B 90, C -94.899, E1 0, E2 0, E3 0, E4 0} C_DIS
LIN {X 295.205, Y 52.102, Z 209.546, A 0, B 90, C -94.814, E1 0, E2 0, E3 0, E4 0} C_DIS
LIN {X 296.057, Y 51.017, Z 210.033, A 0, B 90, C -94.727, E1 0, E2 0, E3 0, E4 0} C_DIS
LIN {X 296.914, Y 49.937, Z 210.523, A 0, B 90, C -94.64, E1 0, E2 0, E3 0, E4 0} C_DIS
LIN {X 297.776, Y 48.863, Z 211.017, A 0, B 90, C -94.552, E1 0, E2 0, E3 0, E4 0} C_DIS
LIN {X 298.643, Y 47.794, Z 211.513, A 0, B 90, C -94.463, E1 0, E2 0, E3 0, E4 0} C_DIS
LIN {X 299.515, Y 46.73, Z 212.012, A 0, B 90, C -94.372, E1 0, E2 0, E3 0, E4 0} C_DIS
LIN {X 300.392, Y 45.672, Z 212.514, A 0, B 90, C -94.281, E1 0, E2 0, E3 0, E4 0} C_DIS
LIN {X 301.274, Y 44.62, Z 213.019, A 0, B 90, C -94.189, E1 0, E2 0, E3 0, E4 0} C_DIS
LIN {X 302.162, Y 43.573, Z 213.526, A 0, B 90, C -94.095, E1 0, E2 0, E3 0, E4 0} C_DIS
LIN {X 303.054, Y 42.532, Z 214.037, A 0, B 90, C -94.001, E1 0, E2 0, E3 0, E4 0} C_DIS
LIN {X 303.951, Y 41.496, Z 214.55, A 0, B 90, C -93.905, E1 0, E2 0, E3 0, E4 0} C_DIS
LIN {X 304.853, Y 40.466, Z 215.066, A 0, B 90, C -93.809, E1 0, E2 0, E3 0, E4 0} C_DIS
LIN {X 305.759, Y 39.442, Z 215.585, A 0, B 90, C -93.711, E1 0, E2 0, E3 0, E4 0} C_DIS
LIN {X 306.671, Y 38.424, Z 216.106, A 0, B 90, C -93.613, E1 0, E2 0, E3 0, E4 0} C_DIS
LIN {X 307.587, Y 37.411, Z 216.631, A 0, B 90, C -93.513, E1 0, E2 0, E3 0, E4 0} C_DIS
LIN {X 308.509, Y 36.404, Z 217.158, A 0, B 90, C -93.412, E1 0, E2 0, E3 0, E4 0} C_DIS
LIN {X 309.435, Y 35.402, Z 217.688, A 0, B 90, C -93.311, E1 0, E2 0, E3 0, E4 0} C_DIS
LIN {X 310.365, Y 34.407, Z 218.22, A 0, B 90, C -93.208, E1 0, E2 0, E3 0, E4 0} C_DIS
LIN {X 311.301, Y 33.418, Z 218.755, A 0, B 90, C -93.104, E1 0, E2 0, E3 0, E4 0} C_DIS
LIN {X 312.241, Y 32.434, Z 219.293, A 0, B 90, C -93, E1 0, E2 0, E3 0, E4 0} C_DIS
LIN {X 313.186, Y 31.456, Z 219.834, A 0, B 90, C -92.894, E1 0, E2 0, E3 0, E4 0} C_DIS
LIN {X 314.135, Y 30.485, Z 220.377, A 0, B 90, C -92.787, E1 0, E2 0, E3 0, E4 0} C_DIS
LIN {X 315.089, Y 29.519, Z 220.923, A 0, B 90, C -92.679, E1 0, E2 0, E3 0, E4 0} C_DIS
LIN {X 316.047, Y 28.559, Z 221.471, A 0, B 90, C -92.57, E1 0, E2 0, E3 0, E4 0} C_DIS
LIN {X 317.01, Y 27.605, Z 222.022, A 0, B 90, C -92.46, E1 0, E2 0, E3 0, E4 0} C_DIS
LIN {X 317.978, Y 26.658, Z 222.576, A 0, B 90, C -92.349, E1 0, E2 0, E3 0, E4 0} C_DIS
LIN {X 318.95, Y 25.716, Z 223.132, A 0, B 90, C -92.237, E1 0, E2 0, E3 0, E4 0} C_DIS
LIN {X 319.927, Y 24.781, Z 223.691, A 0, B 90, C -92.124, E1 0, E2 0, E3 0, E4 0} C_DIS
LIN {X 320.907, Y 23.852, Z 224.252, A 0, B 90, C -92.01, E1 0, E2 0, E3 0, E4 0} C_DIS
LIN {X 321.893, Y 22.929, Z 224.816, A 0, B 90, C -91.895, E1 0, E2 0, E3 0, E4 0} C_DIS
LIN {X 322.882, Y 22.012, Z 225.382, A 0, B 90, C -91.779, E1 0, E2 0, E3 0, E4 0} C_DIS
LIN {X 323.876, Y 21.101, Z 225.951, A 0, B 90, C -91.662, E1 0, E2 0, E3 0, E4 0} C_DIS
LIN {X 324.875, Y 20.197, Z 226.522, A 0, B 90, C -91.544, E1 0, E2 0, E3 0, E4 0} C_DIS
LIN {X 325.877, Y 19.299, Z 227.096, A 0, B 90, C -91.425, E1 0, E2 0, E3 0, E4 0} C_DIS
LIN {X 326.884, Y 18.407, Z 227.672, A 0, B 90, C -91.305, E1 0, E2 0, E3 0, E4 0} C_DIS
LIN {X 327.895, Y 17.522, Z 228.25, A 0, B 90, C -91.184, E1 0, E2 0, E3 0, E4 0} C_DIS
LIN {X 328.91, Y 16.643, Z 228.831, A 0, B 90, C -91.061, E1 0, E2 0, E3 0, E4 0} C_DIS
LIN {X 329.929, Y 15.77, Z 229.414, A 0, B 90, C -90.938, E1 0, E2 0, E3 0, E4 0} C_DIS
LIN {X 330.953, Y 14.904, Z 230, A 0, B 90, C -90.814, E1 0, E2 0, E3 0, E4 0} C_DIS
LIN {X 331.98, Y 14.044, Z 230.588, A 0, B 90, C -90.689, E1 0, E2 0, E3 0, E4 0} C_DIS
LIN {X 333.012, Y 13.191, Z 231.178, A 0, B 90, C -90.563, E1 0, E2 0, E3 0, E4 0} C_DIS
LIN {X 334.047, Y 12.344, Z 231.77, A 0, B 90, C -90.436, E1 0, E2 0, E3 0, E4 0} C_DIS
LIN {X 335.087, Y 11.504, Z 232.365, A 0, B 90, C -90.308, E1 0, E2 0, E3 0, E4 0} C_DIS
LIN {X 336.131, Y 10.67, Z 232.962, A 0, B 90, C -90.179, E1 0, E2 0, E3 0, E4 0} C_DIS
LIN {X 337.178, Y 9.843, Z 233.562, A 0, B 90, C -90.049, E1 0, E2 0, E3 0, E4 0} C_DIS
LIN {X 338.229, Y 9.022, Z 234.163, A 0, B 90, C -89.918, E1 0, E2 0, E3 0, E4 0} C_DIS
LIN {X 339.285, Y 8.208, Z 234.767, A 0, B 90, C -89.787, E1 0, E2 0, E3 0, E4 0} C_DIS
LIN {X 340.344, Y 7.401, Z 235.373, A 0, B 90, C -89.654, E1 0, E2 0, E3 0, E4 0} C_DIS
LIN {X 341.407, Y 6.601, Z 235.981, A 0, B 90, C -89.52, E1 0, E2 0, E3 0, E4 0} C_DIS
LIN {X 342.473, Y 5.807, Z 236.592, A 0, B 90, C -89.386, E1 0, E2 0, E3 0, E4 0} C_DIS
LIN {X 343.544, Y 5.02, Z 237.204, A 0, B 90, C -89.25, E1 0, E2 0, E3 0, E4 0} C_DIS
LIN {X 344.618, Y 4.239, Z 237.819, A 0, B 90, C -89.114, E1 0, E2 0, E3 0, E4 0} C_DIS
LIN {X 345.696, Y 3.466, Z 238.435, A 0, B 90, C -88.976, E1 0, E2 0, E3 0, E4 0} C_DIS
LIN {X 346.777, Y 2.699, Z 239.054, A 0, B 90, C -88.838, E1 0, E2 0, E3 0, E4 0} C_DIS
LIN {X 347.863, Y 1.939, Z 239.675, A 0, B 90, C -88.699, E1 0, E2 0, E3 0, E4 0} C_DIS
LIN {X 348.951, Y 1.186, Z 240.298, A 0, B 90, C -88.559, E1 0, E2 0, E3 0, E4 0} C_DIS
LIN {X 350.043, Y 0.439, Z 240.923, A 0, B 90, C -88.418, E1 0, E2 0, E3 0, E4 0} C_DIS
LIN {X 351.139, Y -0.3, Z 241.55, A 0, B 90, C -88.276, E1 0, E2 0, E3 0, E4 0} C_DIS
LIN {X 352.239, Y -1.033, Z 242.179, A 0, B 90, C -88.134, E1 0, E2 0, E3 0, E4 0} C_DIS
LIN {X 353.341, Y -1.758, Z 242.81, A 0, B 90, C -87.99, E1 0, E2 0, E3 0, E4 0} C_DIS
LIN {X 354.447, Y -2.477, Z 243.443, A 0, B 90, C -87.846, E1 0, E2 0, E3 0, E4 0} C_DIS
LIN {X 355.557, Y -3.189, Z 244.078, A 0, B 90, C -87.701, E1 0, E2 0, E3 0, E4 0} C_DIS
LIN {X 356.67, Y -3.894, Z 244.714, A 0, B 90, C -87.555, E1 0, E2 0, E3 0, E4 0} C_DIS
LIN {X 357.786, Y -4.591, Z 245.353, A 0, B 90, C -87.408, E1 0, E2 0, E3 0, E4 0} C_DIS
LIN {X 358.905, Y -5.282, Z 245.994, A 0, B 90, C -87.26, E1 0, E2 0, E3 0, E4 0} C_DIS
LIN {X 360.028, Y -5.966, Z 246.636, A 0, B 90, C -87.112, E1 0, E2 0, E3 0, E4 0} C_DIS
LIN {X 361.154, Y -6.642, Z 247.28, A 0, B 90, C -86.963, E1 0, E2 0, E3 0, E4 0} C_DIS
LIN {X 362.283, Y -7.312, Z 247.926, A 0, B 90, C -86.813, E1 0, E2 0, E3 0, E4 0} C_DIS
LIN {X 363.416, Y -7.974, Z 248.574, A 0, B 90, C -86.662, E1 0, E2 0, E3 0, E4 0} C_DIS
LIN {X 364.551, Y -8.629, Z 249.224, A 0, B 90, C -86.511, E1 0, E2 0, E3 0, E4 0} C_DIS
LIN {X 365.69, Y -9.277, Z 249.875, A 0, B 90, C -86.358, E1 0, E2 0, E3 0, E4 0} C_DIS
LIN {X 366.831, Y -9.918, Z 250.528, A 0, B 90, C -86.206, E1 0, E2 0, E3 0, E4 0} C_DIS
LIN {X 367.976, Y -10.552, Z 251.183, A 0, B 90, C -86.052, E1 0, E2 0, E3 0, E4 0} C_DIS
LIN {X 369.123, Y -11.179, Z 251.84, A 0, B 90, C -85.898, E1 0, E2 0, E3 0, E4 0} C_DIS
LIN {X 370.274, Y -11.798, Z 252.498, A 0, B 90, C -85.743, E1 0, E2 0, E3 0, E4 0} C_DIS
LIN {X 371.427, Y -12.41, Z 253.158, A 0, B 90, C -85.587, E1 0, E2 0, E3 0, E4 0} C_DIS
LIN {X 372.584, Y -13.015, Z 253.82, A 0, B 90, C -85.43, E1 0, E2 0, E3 0, E4 0} C_DIS
LIN {X 373.743, Y -13.612, Z 254.483, A 0, B 90, C -85.273, E1 0, E2 0, E3 0, E4 0} C_DIS
LIN {X 374.905, Y -14.202, Z 255.148, A 0, B 90, C -85.116, E1 0, E2 0, E3 0, E4 0} C_DIS
LIN {X 376.07, Y -14.785, Z 255.814, A 0, B 90, C -84.957, E1 0, E2 0, E3 0, E4 0} C_DIS
LIN {X 377.237, Y -15.361, Z 256.482, A 0, B 90, C -84.798, E1 0, E2 0, E3 0, E4 0} C_DIS
LIN {X 378.407, Y -15.929, Z 257.152, A 0, B 90, C -84.639, E1 0, E2 0, E3 0, E4 0} C_DIS
LIN {X 379.58, Y -16.49, Z 257.823, A 0, B 90, C -84.479, E1 0, E2 0, E3 0, E4 0} C_DIS
LIN {X 380.756, Y -17.043, Z 258.496, A 0, B 90, C -84.318, E1 0, E2 0, E3 0, E4 0} C_DIS
LIN {X 381.934, Y -17.589, Z 259.17, A 0, B 90, C -84.157, E1 0, E2 0, E3 0, E4 0} C_DIS
LIN {X 383.115, Y -18.128, Z 259.845, A 0, B 90, C -83.995, E1 0, E2 0, E3 0, E4 0} C_DIS
LIN {X 384.298, Y -18.659, Z 260.522, A 0, B 90, C -83.833, E1 0, E2 0, E3 0, E4 0} C_DIS
LIN {X 385.484, Y -19.183, Z 261.201, A 0, B 90, C -83.67, E1 0, E2 0, E3 0, E4 0} C_DIS
LIN {X 386.672, Y -19.699, Z 261.881, A 0, B 90, C -83.506, E1 0, E2 0, E3 0, E4 0} C_DIS
LIN {X 387.862, Y -20.208, Z 262.562, A 0, B 90, C -83.342, E1 0, E2 0, E3 0, E4 0} C_DIS
LIN {X 389.055, Y -20.709, Z 263.245, A 0, B 90, C -83.178, E1 0, E2 0, E3 0, E4 0} C_DIS
LIN {X 390.251, Y -21.203, Z 263.929, A 0, B 90, C -83.013, E1 0, E2 0, E3 0, E4 0} C_DIS
LIN {X 391.449, Y -21.689, Z 264.614, A 0, B 90, C -82.848, E1 0, E2 0, E3 0, E4 0} C_DIS
LIN {X 392.649, Y -22.168, Z 265.301, A 0, B 90, C -82.682, E1 0, E2 0, E3 0, E4 0} C_DIS
LIN {X 393.851, Y -22.639, Z 265.988, A 0, B 90, C -82.516, E1 0, E2 0, E3 0, E4 0} C_DIS
LIN {X 395.055, Y -23.103, Z 266.678, A 0, B 90, C -82.35, E1 0, E2 0, E3 0, E4 0} C_DIS
LIN {X 396.262, Y -23.559, Z 267.368, A 0, B 90, C -82.183, E1 0, E2 0, E3 0, E4 0} C_DIS
LIN {X 397.471, Y -24.007, Z 268.06, A 0, B 90, C -82.016, E1 0, E2 0, E3 0, E4 0} C_DIS
LIN {X 398.682, Y -24.448, Z 268.753, A 0, B 90, C -81.848, E1 0, E2 0, E3 0, E4 0} C_DIS
LIN {X 399.895, Y -24.881, Z 269.447, A 0, B 90, C -81.68, E1 0, E2 0, E3 0, E4 0} C_DIS
LIN {X 401.11, Y -25.307, Z 270.142, A 0, B 90, C -81.512, E1 0, E2 0, E3 0, E4 0} C_DIS
LIN {X 402.327, Y -25.725, Z 270.838, A 0, B 90, C -81.344, E1 0, E2 0, E3 0, E4 0} C_DIS
LIN {X 403.546, Y -26.135, Z 271.536, A 0, B 90, C -81.175, E1 0, E2 0, E3 0, E4 0} C_DIS
LIN {X 404.766, Y -26.538, Z 272.234, A 0, B 90, C -81.006, E1 0, E2 0, E3 0, E4 0} C_DIS
LIN {X 405.989, Y -26.933, Z 272.934, A 0, B 90, C -80.836, E1 0, E2 0, E3 0, E4 0} C_DIS
LIN {X 407.214, Y -27.32, Z 273.634, A 0, B 90, C -80.667, E1 0, E2 0, E3 0, E4 0} C_DIS
LIN {X 408.44, Y -27.699, Z 274.336, A 0, B 90, C -80.497, E1 0, E2 0, E3 0, E4 0} C_DIS
LIN {X 409.668, Y -28.071, Z 275.039, A 0, B 90, C -80.327, E1 0, E2 0, E3 0, E4 0} C_DIS
LIN {X 410.898, Y -28.435, Z 275.743, A 0, B 90, C -80.157, E1 0, E2 0, E3 0, E4 0} C_DIS
LIN {X 412.13, Y -28.791, Z 276.447, A 0, B 90, C -79.987, E1 0, E2 0, E3 0, E4 0} C_DIS
LIN {X 413.363, Y -29.14, Z 277.153, A 0, B 90, C -79.816, E1 0, E2 0, E3 0, E4 0} C_DIS
LIN {X 414.598, Y -29.481, Z 277.86, A 0, B 90, C -79.646, E1 0, E2 0, E3 0, E4 0} C_DIS
LIN {X 415.835, Y -29.814, Z 278.567, A 0, B 90, C -79.475, E1 0, E2 0, E3 0, E4 0} C_DIS
LIN {X 417.073, Y -30.139, Z 279.276, A 0, B 90, C -79.304, E1 0, E2 0, E3 0, E4 0} C_DIS
LIN {X 418.313, Y -30.456, Z 279.985, A 0, B 90, C -79.133, E1 0, E2 0, E3 0, E4 0} C_DIS
LIN {X 419.554, Y -30.766, Z 280.695, A 0, B 90, C -78.962, E1 0, E2 0, E3 0, E4 0} C_DIS
LIN {X 420.797, Y -31.068, Z 281.406, A 0, B 90, C -78.791, E1 0, E2 0, E3 0, E4 0} C_DIS
LIN {X 422.04, Y -31.362, Z 282.118, A 0, B 90, C -78.621, E1 0, E2 0, E3 0, E4 0} C_DIS
LIN {X 423.286, Y -31.648, Z 282.83, A 0, B 90, C -78.45, E1 0, E2 0, E3 0, E4 0} C_DIS
LIN {X 424.533, Y -31.926, Z 283.544, A 0, B 90, C -78.279, E1 0, E2 0, E3 0, E4 0} C_DIS
LIN {X 425.781, Y -32.197, Z 284.258, A 0, B 90, C -78.108, E1 0, E2 0, E3 0, E4 0} C_DIS
LIN {X 427.03, Y -32.459, Z 284.973, A 0, B 90, C -77.937, E1 0, E2 0, E3 0, E4 0} C_DIS
LIN {X 428.28, Y -32.714, Z 285.688, A 0, B 90, C -77.766, E1 0, E2 0, E3 0, E4 0} C_DIS
LIN {X 429.532, Y -32.961, Z 286.404, A 0, B 90, C -77.595, E1 0, E2 0, E3 0, E4 0} C_DIS
LIN {X 430.785, Y -33.2, Z 287.121, A 0, B 90, C -77.425, E1 0, E2 0, E3 0, E4 0} C_DIS
LIN {X 432.039, Y -33.431, Z 287.839, A 0, B 90, C -77.254, E1 0, E2 0, E3 0, E4 0} C_DIS
LIN {X 433.294, Y -33.655, Z 288.557, A 0, B 90, C -77.084, E1 0, E2 0, E3 0, E4 0} C_DIS
LIN {X 434.55, Y -33.87, Z 289.275, A 0, B 90, C -76.913, E1 0, E2 0, E3 0, E4 0} C_DIS
LIN {X 435.807, Y -34.077, Z 289.995, A 0, B 90, C -76.743, E1 0, E2 0, E3 0, E4 0} C_DIS
LIN {X 437.065, Y -34.277, Z 290.715, A 0, B 90, C -76.574, E1 0, E2 0, E3 0, E4 0} C_DIS
LIN {X 438.324, Y -34.469, Z 291.435, A 0, B 90, C -76.404, E1 0, E2 0, E3 0, E4 0} C_DIS
LIN {X 439.584, Y -34.652, Z 292.156, A 0, B 90, C -76.234, E1 0, E2 0, E3 0, E4 0} C_DIS
LIN {X 440.845, Y -34.828, Z 292.877, A 0, B 90, C -76.065, E1 0, E2 0, E3 0, E4 0} C_DIS
LIN {X 442.106, Y -34.996, Z 293.599, A 0, B 90, C -75.896, E1 0, E2 0, E3 0, E4 0} C_DIS
LIN {X 443.368, Y -35.156, Z 294.321, A 0, B 90, C -75.728, E1 0, E2 0, E3 0, E4 0} C_DIS
LIN {X 444.631, Y -35.308, Z 295.044, A 0, B 90, C -75.559, E1 0, E2 0, E3 0, E4 0} C_DIS
LIN {X 445.895, Y -35.452, Z 295.767, A 0, B 90, C -75.391, E1 0, E2 0, E3 0, E4 0} C_DIS
LIN {X 447.159, Y -35.588, Z 296.49, A 0, B 90, C -75.224, E1 0, E2 0, E3 0, E4 0} C_DIS
LIN {X 448.424, Y -35.716, Z 297.214, A 0, B 90, C -75.056, E1 0, E2 0, E3 0, E4 0} C_DIS
LIN {X 449.69, Y -35.836, Z 297.938, A 0, B 90, C -74.889, E1 0, E2 0, E3 0, E4 0} C_DIS
LIN {X 450.956, Y -35.949, Z 298.663, A 0, B 90, C -74.722, E1 0, E2 0, E3 0, E4 0} C_DIS
LIN {X 452.223, Y -36.053, Z 299.388, A 0, B 90, C -74.556, E1 0, E2 0, E3 0, E4 0} C_DIS
LIN {X 453.49, Y -36.149, Z 300.113, A 0, B 90, C -74.39, E1 0, E2 0, E3 0, E4 0} C_DIS
LIN {X 454.758, Y -36.237, Z 300.838, A 0, B 90, C -74.225, E1 0, E2 0, E3 0, E4 0} C_DIS
LIN {X 456.026, Y -36.318, Z 301.563, A 0, B 90, C -74.06, E1 0, E2 0, E3 0, E4 0} C_DIS
LIN {X 457.294, Y -36.39, Z 302.289, A 0, B 90, C -73.895, E1 0, E2 0, E3 0, E4 0} C_DIS
LIN {X 458.563, Y -36.455, Z 303.015, A 0, B 90, C -73.731, E1 0, E2 0, E3 0, E4 0} C_DIS
LIN {X 459.832, Y -36.511, Z 303.741, A 0, B 90, C -73.568, E1 0, E2 0, E3 0, E4 0} C_DIS
LIN {X 461.101, Y -36.559, Z 304.467, A 0, B 90, C -73.405, E1 0, E2 0, E3 0, E4 0} C_DIS
LIN {X 462.37, Y -36.6, Z 305.194, A 0, B 90, C -73.242, E1 0, E2 0, E3 0, E4 0} C_DIS
LIN {X 463.64, Y -36.632, Z 305.92, A 0, B 90, C -73.08, E1 0, E2 0, E3 0, E4 0} C_DIS
LIN {X 464.91, Y -36.657, Z 306.646, A 0, B 90, C -72.918, E1 0, E2 0, E3 0, E4 0} C_DIS
LIN {X 466.179, Y -36.673, Z 307.373, A 0, B 90, C -72.758, E1 0, E2 0, E3 0, E4 0} C_DIS
LIN {X 467.449, Y -36.682, Z 308.1, A 0, B 90, C -72.597, E1 0, E2 0, E3 0, E4 0} C_DIS
LIN {X 468.719, Y -36.682, Z 308.826, A 0, B 90, C -72.437, E1 0, E2 0, E3 0, E4 0} C_DIS
LIN {X 469.989, Y -36.675, Z 309.553, A 0, B 90, C -72.278, E1 0, E2 0, E3 0, E4 0} C_DIS
LIN {X 471.259, Y -36.659, Z 310.279, A 0, B 90, C -72.12, E1 0, E2 0, E3 0, E4 0} C_DIS
LIN {X 472.529, Y -36.636, Z 311.006, A 0, B 90, C -71.962, E1 0, E2 0, E3 0, E4 0} C_DIS
LIN {X 473.798, Y -36.604, Z 311.732, A 0, B 90, C -71.805, E1 0, E2 0, E3 0, E4 0} C_DIS
LIN {X 475.068, Y -36.565, Z 312.459, A 0, B 90, C -71.648, E1 0, E2 0, E3 0, E4 0} C_DIS
LIN {X 476.337, Y -36.518, Z 313.185, A 0, B 90, C -71.492, E1 0, E2 0, E3 0, E4 0} C_DIS
LIN {X 477.606, Y -36.462, Z 313.911, A 0, B 90, C -71.337, E1 0, E2 0, E3 0, E4 0} C_DIS
LIN {X 478.875, Y -36.399, Z 314.637, A 0, B 90, C -71.182, E1 0, E2 0, E3 0, E4 0} C_DIS
LIN {X 480.143, Y -36.328, Z 315.363, A 0, B 90, C -71.028, E1 0, E2 0, E3 0, E4 0} C_DIS
LIN {X 481.411, Y -36.248, Z 316.088, A 0, B 90, C -70.875, E1 0, E2 0, E3 0, E4 0} C_DIS
LIN {X 482.679, Y -36.161, Z 316.814, A 0, B 90, C -70.723, E1 0, E2 0, E3 0, E4 0} C_DIS
LIN {X 483.946, Y -36.066, Z 317.539, A 0, B 90, C -70.571, E1 0, E2 0, E3 0, E4 0} C_DIS
LIN {X 485.213, Y -35.962, Z 318.263, A 0, B 90, C -70.42, E1 0, E2 0, E3 0, E4 0} C_DIS
LIN {X 486.479, Y -35.851, Z 318.988, A 0, B 90, C -70.27, E1 0, E2 0, E3 0, E4 0} C_DIS
LIN {X 487.745, Y -35.732, Z 319.712, A 0, B 90, C -70.121, E1 0, E2 0, E3 0, E4 0} C_DIS
LIN {X 489.01, Y -35.605, Z 320.436, A 0, B 90, C -69.972, E1 0, E2 0, E3 0, E4 0} C_DIS
LIN {X 490.274, Y -35.47, Z 321.159, A 0, B 90, C -69.824, E1 0, E2 0, E3 0, E4 0} C_DIS
LIN {X 491.538, Y -35.327, Z 321.883, A 0, B 90, C -69.677, E1 0, E2 0, E3 0, E4 0} C_DIS
LIN {X 492.801, Y -35.176, Z 322.605, A 0, B 90, C -69.531, E1 0, E2 0, E3 0, E4 0} C_DIS
LIN {X 494.063, Y -35.017, Z 323.328, A 0, B 90, C -69.386, E1 0, E2 0, E3 0, E4 0} C_DIS
LIN {X 495.325, Y -34.85, Z 324.049, A 0, B 90, C -69.242, E1 0, E2 0, E3 0, E4 0} C_DIS
LIN {X 496.586, Y -34.675, Z 324.771, A 0, B 90, C -69.098, E1 0, E2 0, E3 0, E4 0} C_DIS
LIN {X 497.846, Y -34.493, Z 325.492, A 0, B 90, C -68.955, E1 0, E2 0, E3 0, E4 0} C_DIS
LIN {X 499.105, Y -34.302, Z 326.212, A 0, B 90, C -68.813, E1 0, E2 0, E3 0, E4 0} C_DIS
LIN {X 500.363, Y -34.104, Z 326.932, A 0, B 90, C -68.672, E1 0, E2 0, E3 0, E4 0} C_DIS
LIN {X 501.62, Y -33.897, Z 327.651, A 0, B 90, C -68.532, E1 0, E2 0, E3 0, E4 0} C_DIS
LIN {X 502.876, Y -33.683, Z 328.37, A 0, B 90, C -68.393, E1 0, E2 0, E3 0, E4 0} C_DIS
LIN {X 504.132, Y -33.46, Z 329.088, A 0, B 90, C -68.255, E1 0, E2 0, E3 0, E4 0} C_DIS
LIN {X 505.386, Y -33.23, Z 329.806, A 0, B 90, C -68.117, E1 0, E2 0, E3 0, E4 0} C_DIS
LIN {X 506.639, Y -32.992, Z 330.523, A 0, B 90, C -67.981, E1 0, E2 0, E3 0, E4 0} C_DIS
LIN {X 507.891, Y -32.746, Z 331.239, A 0, B 90, C -67.845, E1 0, E2 0, E3 0, E4 0} C_DIS
LIN {X 509.141, Y -32.493, Z 331.955, A 0, B 90, C -67.711, E1 0, E2 0, E3 0, E4 0} C_DIS
LIN {X 510.391, Y -32.231, Z 332.67, A 0, B 90, C -67.577, E1 0, E2 0, E3 0, E4 0} C_DIS
LIN {X 511.639, Y -31.961, Z 333.384, A 0, B 90, C -67.444, E1 0, E2 0, E3 0, E4 0} C_DIS
LIN {X 512.886, Y -31.684, Z 334.097, A 0, B 90, C -67.313, E1 0, E2 0, E3 0, E4 0} C_DIS
LIN {X 514.131, Y -31.399, Z 334.81, A 0, B 90, C -67.182, E1 0, E2 0, E3 0, E4 0} C_DIS
LIN {X 515.375, Y -31.106, Z 335.522, A 0, B 90, C -67.052, E1 0, E2 0, E3 0, E4 0} C_DIS
LIN {X 516.618, Y -30.805, Z 336.233, A 0, B 90, C -66.923, E1 0, E2 0, E3 0, E4 0} C_DIS
LIN {X 517.859, Y -30.496, Z 336.943, A 0, B 90, C -66.795, E1 0, E2 0, E3 0, E4 0} C_DIS
LIN {X 519.099, Y -30.18, Z 337.652, A 0, B 90, C -66.669, E1 0, E2 0, E3 0, E4 0} C_DIS
LIN {X 520.338, Y -29.856, Z 338.361, A 0, B 90, C -66.543, E1 0, E2 0, E3 0, E4 0} C_DIS
LIN {X 521.574, Y -29.524, Z 339.069, A 0, B 90, C -66.418, E1 0, E2 0, E3 0, E4 0} C_DIS
